C07252=1043.907,204.076,-99.284,170.932,38.862,157.345
C07253=1043.914,204.324,-99.309,170.935,38.863,157.345
C07254=1043.920,204.573,-99.334,170.938,38.865,157.345
C07255=1043.927,204.821,-99.359,170.940,38.867,157.346
C07256=1043.933,205.071,-99.384,170.943,38.868,157.346
C07257=1043.959,206.122,-99.491,171.208,38.971,157.375
C07258=1043.966,206.407,-99.521,171.211,38.973,157.375
C07259=1043.974,206.692,-99.551,171.213,38.976,157.376
C07260=1043.982,206.977,-99.581,171.216,38.979,157.376
C07261=1043.989,207.263,-99.612,171.219,38.982,157.377
C07262=1043.995,207.512,-99.637,171.220,38.984,157.378
C07263=1044.003,207.760,-99.664,171.223,38.987,157.378
C07264=1044.008,208.009,-99.690,171.224,38.989,157.379
C07265=1044.015,208.257,-99.717,171.227,38.992,157.379
C07266=1044.022,208.505,-99.743,171.229,38.994,157.380
C07267=1044.028,208.755,-99.770,171.231,38.997,157.381
C07268=1044.035,209.003,-99.796,171.234,38.999,157.381
C07269=1044.042,209.251,-99.822,171.235,39.002,157.382
C07270=1044.048,209.500,-99.849,171.238,39.004,157.382
C07271=1044.055,209.748,-99.875,171.239,39.007,157.383
C07272=1044.061,209.996,-99.901,171.242,39.009,157.384
C07273=1044.068,210.245,-99.929,171.244,39.012,157.384
C07274=1044.075,210.493,-99.955,171.246,39.014,157.385
C07275=1044.082,210.742,-99.982,171.248,39.017,157.385
C07276=1044.087,210.990,-100.008,171.250,39.019,157.386
C07277=1044.095,211.239,-100.035,171.252,39.022,157.386
C07278=1044.101,211.488,-100.062,171.255,39.024,157.387
C07279=1044.107,211.736,-100.088,171.256,39.027,157.388
C07280=1044.115,211.985,-100.114,171.259,39.029,157.388
C07281=1044.120,212.233,-100.141,171.262,39.032,157.389
C07282=1044.127,212.481,-100.169,171.263,39.035,157.389
C07283=1044.133,212.730,-100.195,171.266,39.037,157.390
C07284=1044.140,212.979,-100.222,171.267,39.039,157.390
C07285=1044.147,213.227,-100.248,171.270,39.042,157.391
C07286=1044.153,213.476,-100.275,171.272,39.044,157.392
C07287=1044.160,213.724,-100.302,171.274,39.047,157.392
C07288=1044.166,213.972,-100.329,171.276,39.049,157.393
C07289=1044.173,214.221,-100.355,171.279,39.052,157.393
C07290=1044.179,214.469,-100.382,171.280,39.054,157.394
C07291=1044.186,214.718,-100.409,171.283,39.057,157.395
C07292=1044.193,214.967,-100.436,171.286,39.059,157.395
C07293=1044.198,215.215,-100.462,171.287,39.062,157.396
C07294=1044.206,215.464,-100.489,171.290,39.064,157.396
C07295=1044.212,215.712,-100.517,171.291,39.067,157.397
C07296=1044.219,215.960,-100.543,171.294,39.069,157.397
C07297=1044.225,216.209,-100.570,171.296,39.072,157.398
C07298=1044.232,216.458,-100.597,171.298,39.074,157.399
C07299=1044.238,216.706,-100.623,171.300,39.077,157.399
C07300=1044.245,216.955,-100.650,171.303,39.079,157.400
C07301=1044.251,217.202,-100.677,171.306,39.082,157.400
C07302=1044.258,217.451,-100.704,171.307,39.084,157.401
C07303=1044.265,217.700,-100.732,171.310,39.087,157.402
C07304=1044.272,217.948,-100.758,171.312,39.089,157.402
C07305=1044.277,218.197,-100.785,171.314,39.091,157.403
C07306=1044.285,218.445,-100.812,171.316,39.094,157.403
C07307=1044.291,218.694,-100.839,171.319,39.096,157.404
C07308=1044.298,218.941,-100.866,171.320,39.099,157.404
C07309=1044.304,219.190,-100.893,171.323,39.101,157.405
C07310=1044.311,219.439,-100.921,171.325,39.103,157.406
C07311=1044.318,219.688,-100.947,171.328,39.106,157.406
C07312=1044.324,219.936,-100.974,171.329,39.109,157.407
C07313=1044.331,220.184,-101.001,171.332,39.111,157.407
C07314=1044.338,220.475,-101.033,171.335,39.114,157.408
C07315=1044.346,220.766,-101.065,171.337,39.117,157.409
C07316=1044.353,221.056,-101.097,171.340,39.120,157.409
C07317=1044.362,221.347,-101.129,171.343,39.123,157.410
C07318=1044.367,221.596,-101.155,171.345,39.125,157.411
C07319=1044.374,221.844,-101.183,171.347,39.128,157.411
C07320=1044.381,222.093,-101.210,171.349,39.130,157.412
C07321=1044.387,222.341,-101.237,171.352,39.133,157.412
C07322=1044.394,222.589,-101.265,171.354,39.135,157.413
C07323=1044.400,222.838,-101.292,171.356,39.138,157.414
C07324=1044.407,223.087,-101.319,171.358,39.140,157.414
C07325=1044.413,223.334,-101.347,171.361,39.142,157.415
C07326=1044.420,223.583,-101.374,171.364,39.145,157.415
C07327=1044.427,223.831,-101.401,171.365,39.148,157.416
C07328=1044.434,224.080,-101.429,171.368,39.150,157.417
C07329=1044.439,224.328,-101.455,171.370,39.152,157.417
C07330=1044.446,224.577,-101.483,171.373,39.155,157.418
C07331=1044.453,224.825,-101.511,171.374,39.158,157.418
C07332=1044.459,225.074,-101.539,171.377,39.160,157.419
C07333=1044.466,225.323,-101.566,171.379,39.162,157.420
C07334=1044.472,225.570,-101.593,171.382,39.164,157.420
C07335=1044.479,225.819,-101.620,171.385,39.167,157.421
C07336=1044.486,226.067,-101.648,171.386,39.170,157.421
C07337=1044.492,226.316,-101.675,171.389,39.172,157.422
C07338=1044.499,226.564,-101.703,171.391,39.174,157.422
C07339=1044.506,226.813,-101.730,171.394,39.177,157.423
C07340=1044.512,227.061,-101.758,171.396,39.179,157.424
C07341=1044.519,227.309,-101.785,171.398,39.182,157.424
C07342=1044.525,227.558,-101.812,171.400,39.184,157.425
C07343=1044.532,227.807,-101.840,171.403,39.186,157.425
C07344=1044.539,228.055,-101.867,171.405,39.189,157.426
C07345=1044.546,228.303,-101.895,171.408,39.192,157.427
C07346=1044.552,228.552,-101.923,171.410,39.194,157.427
C07347=1044.559,228.800,-101.950,171.412,39.196,157.428
C07348=1044.565,229.048,-101.978,171.415,39.199,157.428
C07349=1044.572,229.296,-102.006,171.417,39.201,157.429
C07350=1044.578,229.545,-102.034,171.420,39.204,157.429
C07351=1044.584,229.793,-102.062,171.421,39.206,157.430
C07352=1044.591,230.042,-102.089,171.424,39.208,157.431
C07353=1044.598,230.290,-102.117,171.427,39.211,157.431
C07354=1044.604,230.539,-102.145,171.429,39.214,157.432
C07355=1044.611,230.786,-102.172,171.432,39.216,157.432
C07356=1044.617,231.035,-102.200,171.434,39.218,157.433
C07357=1044.624,231.283,-102.228,171.436,39.221,157.434
C07358=1044.631,231.532,-102.255,171.438,39.223,157.434
C07359=1044.637,231.781,-102.284,171.441,39.226,157.435
C07360=1044.643,232.029,-102.311,171.443,39.228,157.435
C07361=1044.650,232.277,-102.339,171.446,39.231,157.436
C07362=1044.657,232.526,-102.367,171.449,39.233,157.437
C07363=1044.663,232.774,-102.395,171.451,39.236,157.437
C07364=1044.669,233.023,-102.423,171.453,39.238,157.438
C07365=1044.675,233.271,-102.450,171.455,39.241,157.438
C07366=1044.682,233.519,-102.479,171.458,39.243,157.439
C07367=1044.689,233.767,-102.506,171.461,39.246,157.440
C07368=1044.695,234.016,-102.535,171.463,39.248,157.440
C07369=1044.702,234.264,-102.562,171.466,39.251,157.441
C07370=1044.709,234.547,-102.595,171.468,39.253,157.441
C07371=1044.717,234.831,-102.627,171.471,39.256,157.442
C07372=1044.724,235.114,-102.658,171.474,39.259,157.443
C07373=1044.731,235.397,-102.691,171.476,39.262,157.444
C07374=1044.738,235.646,-102.718,171.479,39.264,157.444
C07375=1044.745,235.894,-102.746,171.481,39.267,157.445
C07376=1044.751,236.142,-102.775,171.484,39.269,157.445
C07377=1044.758,236.391,-102.803,171.487,39.272,157.446
C07378=1044.764,236.639,-102.831,171.489,39.274,157.447
C07379=1044.771,236.887,-102.858,171.492,39.276,157.447
C07380=1044.777,237.136,-102.887,171.494,39.279,157.448
C07381=1044.784,237.384,-102.915,171.497,39.282,157.448
C07382=1044.790,237.632,-102.943,171.498,39.284,157.449
C07383=1044.797,237.881,-102.972,171.501,39.286,157.449
C07384=1044.803,238.129,-103.000,171.504,39.289,157.450
C07385=1044.810,238.377,-103.028,171.506,39.291,157.451
C07386=1044.816,238.626,-103.056,171.509,39.294,157.451
C07387=1044.823,238.874,-103.084,171.511,39.296,157.452
C07388=1044.830,239.122,-103.113,171.514,39.299,157.453
C07389=1044.837,239.371,-103.141,171.516,39.301,157.453
C07390=1044.844,239.619,-103.170,171.519,39.303,157.454
C07391=1044.850,239.868,-103.197,171.521,39.306,157.454
C07392=1044.856,240.116,-103.226,171.524,39.309,157.455
C07393=1044.863,240.364,-103.254,171.527,39.311,157.455
C07394=1044.870,240.613,-103.282,171.529,39.313,157.456
C07395=1044.876,240.861,-103.311,171.532,39.315,157.457
C07396=1044.883,241.109,-103.339,171.534,39.318,157.457
C07397=1044.889,241.357,-103.368,171.537,39.321,157.458
C07398=1044.896,241.606,-103.395,171.540,39.323,157.458
C07399=1044.902,241.854,-103.425,171.542,39.326,157.459
C07400=1044.909,242.102,-103.453,171.545,39.328,157.460
C07401=1044.915,242.350,-103.481,171.547,39.330,157.460
C07402=1044.922,242.599,-103.511,171.550,39.333,157.461
C07403=1044.929,242.847,-103.539,171.553,39.335,157.462
C07404=1044.935,243.096,-103.567,171.554,39.338,157.462
C07405=1044.942,243.344,-103.596,171.557,39.341,157.463
C07406=1044.948,243.592,-103.624,171.559,39.343,157.463
C07407=1044.954,243.841,-103.653,171.562,39.345,157.464
C07408=1044.961,244.088,-103.682,171.564,39.348,157.465
C07409=1044.967,244.336,-103.711,171.567,39.350,157.465
C07410=1044.974,244.585,-103.738,171.570,39.353,157.466
C07411=1044.981,244.834,-103.768,171.572,39.355,157.466
C07412=1044.987,245.082,-103.797,171.575,39.358,157.467
C07413=1044.994,245.330,-103.825,171.577,39.360,157.468
C07414=1045.000,245.578,-103.854,171.580,39.363,157.468
C07415=1045.006,245.827,-103.883,171.583,39.365,157.469
C07416=1045.012,246.075,-103.912,171.585,39.368,157.470
C07417=1045.019,246.323,-103.940,171.588,39.370,157.470
C07418=1045.026,246.571,-103.969,171.590,39.373,157.471
C07419=1045.032,246.820,-103.998,171.593,39.375,157.471
C07420=1045.038,247.068,-104.027,171.596,39.378,157.472
C07421=1045.045,247.316,-104.056,171.598,39.381,157.473
C07422=1045.051,247.565,-104.085,171.601,39.383,157.473
C07423=1045.057,247.813,-104.114,171.603,39.386,157.474
C07424=1045.064,248.060,-104.143,171.606,39.388,157.474
C07425=1045.070,248.309,-104.172,171.610,39.390,157.475
C07426=1045.077,248.587,-104.204,171.612,39.393,157.476
C07427=1045.085,248.864,-104.236,171.615,39.396,157.476
C07428=1045.092,249.141,-104.269,171.618,39.399,157.477
C07429=1045.099,249.419,-104.302,171.621,39.402,157.478
C07430=1045.106,249.667,-104.330,171.624,39.405,157.479
C07431=1045.112,249.915,-104.359,171.627,39.407,157.479
C07432=1045.119,250.164,-104.389,171.629,39.409,157.480
C07433=1045.125,250.412,-104.418,171.632,39.412,157.480
C07434=1045.131,250.660,-104.447,171.634,39.414,157.481
C07435=1045.137,250.908,-104.476,171.637,39.417,157.482
C07436=1045.144,251.157,-104.505,171.640,39.419,157.482
C07437=1045.151,251.405,-104.534,171.642,39.422,157.483
C07438=1045.157,251.653,-104.563,171.645,39.424,157.484
C07439=1045.164,251.900,-104.592,171.647,39.427,157.484
C07440=1045.171,252.149,-104.622,171.650,39.430,157.485
C07441=1045.177,252.397,-104.651,171.654,39.432,157.485
C07442=1045.183,252.646,-104.680,171.656,39.434,157.486
C07443=1045.190,252.894,-104.709,171.659,39.437,157.487
C07444=1045.197,253.143,-104.738,171.661,39.439,157.487
C07445=1045.203,253.391,-104.767,171.664,39.442,157.488
C07446=1045.209,253.639,-104.796,171.667,39.444,157.488
C07447=1045.216,253.887,-104.826,171.669,39.447,157.489
C07448=1045.222,254.135,-104.855,171.672,39.449,157.490
C07449=1045.229,254.383,-104.885,171.674,39.452,157.490
C07450=1045.236,254.632,-104.913,171.678,39.454,157.491
C07451=1045.243,254.879,-104.943,171.681,39.457,157.492
C07452=1045.249,255.127,-104.972,171.683,39.459,157.492
C07453=1045.256,255.376,-105.002,171.686,39.462,157.493
C07454=1045.262,255.624,-105.031,171.688,39.464,157.493
C07455=1045.269,255.872,-105.060,171.691,39.466,157.494
C07456=1045.276,256.121,-105.090,171.694,39.469,157.495
C07457=1045.282,256.369,-105.119,171.697,39.471,157.495
C07458=1045.289,256.618,-105.148,171.700,39.474,157.496
C07459=1045.295,256.865,-105.178,171.702,39.477,157.497
C07460=1045.302,257.113,-105.207,171.705,39.479,157.497
C07461=1045.308,257.362,-105.236,171.708,39.482,157.498
C07462=1045.315,257.610,-105.266,171.710,39.484,157.498
C07463=1045.322,257.859,-105.296,171.714,39.486,157.499
C07464=1045.329,258.106,-105.325,171.717,39.489,157.500
C07465=1045.335,258.354,-105.354,171.719,39.491,157.500
C07466=1045.342,258.603,-105.383,171.722,39.494,157.501
C07467=1045.349,258.850,-105.413,171.724,39.496,157.502
C07468=1045.356,259.099,-105.442,171.728,39.498,157.502
C07469=1045.362,259.347,-105.472,171.731,39.501,157.503
C07470=1045.369,259.595,-105.501,171.733,39.504,157.503
C07471=1045.376,259.843,-105.531,171.736,39.506,157.504
C07472=1045.382,260.092,-105.561,171.738,39.509,157.505
C07473=1045.389,260.339,-105.590,171.742,39.511,157.505
C07474=1045.396,260.588,-105.620,171.745,39.513,157.506
C07475=1045.402,260.836,-105.650,171.747,39.516,157.507
C07476=1045.409,261.084,-105.679,171.750,39.518,157.507
C07477=1045.416,261.332,-105.709,171.754,39.521,157.508
C07478=1045.423,261.581,-105.738,171.756,39.523,157.508
C07479=1045.429,261.828,-105.768,171.759,39.525,157.509
C07480=1045.436,262.077,-105.797,171.761,39.528,157.510
C07481=1045.443,262.325,-105.827,171.765,39.530,157.510
C07482=1045.450,262.600,-105.860,171.768,39.533,157.511
C07483=1045.457,262.876,-105.894,171.771,39.536,157.512
C07484=1045.465,263.153,-105.926,171.774,39.539,157.513
C07485=1045.472,263.429,-105.960,171.778,39.542,157.513
C07486=1045.479,263.677,-105.990,171.780,39.545,157.514
C07487=1045.485,263.925,-106.020,171.783,39.547,157.515
C07488=1045.492,264.173,-106.050,171.786,39.550,157.515
C07489=1045.498,264.421,-106.079,171.788,39.552,157.516
C07490=1045.505,264.670,-106.110,171.792,39.555,157.517
C07491=1045.511,264.917,-106.140,171.794,39.557,157.517
C07492=1045.518,265.165,-106.170,171.797,39.560,157.518
C07493=1045.524,265.413,-106.200,171.801,39.563,157.519
C07494=1045.531,265.662,-106.230,171.803,39.565,157.519
C07495=1045.537,265.910,-106.259,171.806,39.568,157.520
C07496=1045.544,266.158,-106.290,171.809,39.570,157.520
C07497=1045.551,266.406,-106.320,171.812,39.573,157.521
C07498=1045.558,266.654,-106.350,171.815,39.575,157.522
C07499=1045.564,266.902,-106.381,171.818,39.578,157.522
C07500=1045.571,267.150,-106.411,171.820,39.580,157.523
C07501=1045.578,267.398,-106.441,171.824,39.583,157.524
C07502=1045.584,267.647,-106.471,171.827,39.585,157.524
C07503=1045.591,267.894,-106.501,171.829,39.588,157.525
C07504=1045.597,268.143,-106.532,171.833,39.591,157.526
C07505=1045.604,268.390,-106.562,171.836,39.593,157.526
C07506=1045.610,268.639,-106.592,171.838,39.596,157.527
C07507=1045.617,268.886,-106.622,171.842,39.598,157.528
C07508=1045.623,269.135,-106.653,171.845,39.601,157.528
C07509=1045.630,269.383,-106.683,171.847,39.603,157.529
C07510=1045.636,269.631,-106.713,171.851,39.606,157.530
C07511=1045.643,269.879,-106.743,171.854,39.609,157.530
C07512=1045.650,270.127,-106.774,171.856,39.611,157.531
C07513=1045.656,270.375,-106.804,171.859,39.614,157.532
C07514=1045.663,270.624,-106.835,171.863,39.616,157.532
C07515=1045.670,270.872,-106.865,171.865,39.619,157.533
C07516=1045.676,271.119,-106.896,171.869,39.621,157.534
C07517=1045.683,271.367,-106.926,171.871,39.624,157.534
C07518=1045.689,271.616,-106.957,171.874,39.626,157.535
C07519=1045.696,271.863,-106.986,171.878,39.629,157.536
C07520=1045.702,272.112,-107.017,171.880,39.631,157.536
C07521=1045.709,272.360,-107.048,171.883,39.634,157.537
C07522=1045.716,272.607,-107.078,171.887,39.637,157.538
C07523=1045.722,272.856,-107.109,171.889,39.639,157.538
C07524=1045.729,273.104,-107.140,171.892,39.642,157.539
C07525=1045.735,273.351,-107.170,171.896,39.645,157.540
C07526=1045.742,273.600,-107.201,171.898,39.647,157.540
C07527=1045.748,273.848,-107.232,171.901,39.650,157.541
C07528=1045.755,274.095,-107.262,171.905,39.653,157.542
C07529=1045.762,274.344,-107.293,171.907,39.655,157.542
C07530=1045.768,274.592,-107.323,171.911,39.658,157.543
C07531=1045.775,274.840,-107.354,171.914,39.660,157.544
C07532=1045.781,275.087,-107.385,171.916,39.663,157.544
C07533=1045.788,275.336,-107.415,171.920,39.665,157.545
C07534=1045.794,275.584,-107.447,171.923,39.668,157.546
C07535=1045.802,275.832,-107.477,171.927,39.671,157.547
C07536=1045.808,276.079,-107.508,171.929,39.673,157.547
C07537=1045.814,276.328,-107.539,171.932,39.676,157.548
C07538=1045.825,276.739,-107.590,171.937,39.681,157.549
C07539=1045.832,276.982,-107.620,171.941,39.683,157.550
C07540=1045.838,277.225,-107.650,171.943,39.686,157.550
C07541=1045.845,277.468,-107.681,171.946,39.688,157.551
C07542=1045.851,277.711,-107.711,171.950,39.691,157.552
C07543=1045.858,277.954,-107.742,171.952,39.693,157.552
C07544=1045.865,278.198,-107.772,171.956,39.696,157.553
C07545=1045.871,278.441,-107.802,171.959,39.698,157.554
C07546=1045.877,278.690,-107.833,171.961,39.701,157.554
C07547=1045.884,278.937,-107.864,171.965,39.704,157.555
C07548=1045.891,279.185,-107.895,171.968,39.707,157.556
C07549=1045.897,279.433,-107.926,171.971,39.709,157.557
C07550=1045.904,279.681,-107.957,171.974,39.712,157.557
C07551=1045.911,279.929,-107.989,171.978,39.714,157.558
C07552=1045.917,280.177,-108.019,171.980,39.717,157.559
C07553=1045.923,280.425,-108.050,171.984,39.720,157.559
C07554=1045.930,280.672,-108.082,171.987,39.723,157.560
C07555=1045.937,280.920,-108.113,171.990,39.726,157.561
C07556=1045.943,281.169,-108.144,171.993,39.728,157.561
C07557=1045.950,281.417,-108.175,171.996,39.731,157.562
C07558=1045.957,281.665,-108.207,172.000,39.733,157.563
C07559=1045.963,281.912,-108.238,172.002,39.736,157.564
C07560=1045.969,282.160,-108.270,172.006,39.739,157.564
C07561=1045.976,282.408,-108.301,172.009,39.742,157.565
C07562=1045.982,282.657,-108.332,172.013,39.744,157.566
C07563=1045.989,282.904,-108.363,172.015,39.747,157.566
C07564=1045.995,283.152,-108.395,172.019,39.749,157.567
C07565=1046.002,283.400,-108.426,172.022,39.752,157.568
C07566=1046.009,283.648,-108.458,172.025,39.755,157.568
C07567=1046.016,283.896,-108.489,172.028,39.758,157.569
C07568=1046.022,284.144,-108.521,172.032,39.760,157.570
C07569=1046.029,284.392,-108.552,172.035,39.763,157.571
C07570=1046.036,284.640,-108.584,172.038,39.766,157.571
C07571=1046.043,284.888,-108.615,172.041,39.769,157.572
C07572=1046.049,285.136,-108.646,172.045,39.772,157.573
C07573=1046.056,285.383,-108.678,172.047,39.774,157.573
C07574=1046.063,285.631,-108.709,172.051,39.776,157.574
C07575=1046.069,285.879,-108.741,172.055,39.779,157.575
C07576=1046.076,286.127,-108.772,172.058,39.782,157.576
C07577=1046.083,286.375,-108.804,172.061,39.785,157.576
C07578=1046.090,286.623,-108.835,172.064,39.788,157.577
C07579=1046.096,286.871,-108.866,172.068,39.790,157.578
C07580=1046.103,287.119,-108.898,172.070,39.793,157.579
C07581=1046.110,287.367,-108.929,172.074,39.796,157.579
C07582=1046.116,287.615,-108.961,172.078,39.799,157.580
C07583=1046.123,287.862,-108.993,172.081,39.801,157.581
C07584=1046.130,288.110,-109.025,172.084,39.804,157.581
C07585=1046.136,288.358,-109.056,172.087,39.807,157.582
C07586=1046.142,288.606,-109.088,172.091,39.810,157.583
C07587=1046.149,288.853,-109.120,172.094,39.812,157.584
C07588=1046.156,289.101,-109.152,172.097,39.815,157.584
C07589=1046.163,289.349,-109.183,172.101,39.818,157.585
C07590=1046.169,289.598,-109.215,172.104,39.821,157.586
C07591=1046.176,289.845,-109.248,172.108,39.823,157.587
C07592=1046.182,290.093,-109.279,172.110,39.826,157.587
C07593=1046.189,290.341,-109.310,172.114,39.829,157.588
C07594=1046.197,290.633,-109.348,172.118,39.832,157.589
C07595=1046.205,290.924,-109.387,172.122,39.835,157.590
C07596=1046.212,291.216,-109.424,172.126,39.839,157.591
C07597=1046.220,291.509,-109.462,172.130,39.842,157.592
C07598=1046.227,291.757,-109.494,172.133,39.845,157.592
C07599=1046.234,292.004,-109.526,172.136,39.848,157.593
C07600=1046.240,292.252,-109.558,172.140,39.850,157.594
C07601=1046.247,292.500,-109.590,172.144,39.853,157.595
C07602=1046.254,292.748,-109.621,172.146,39.856,157.595
C07603=1046.260,292.995,-109.654,172.150,39.859,157.596
C07604=1046.268,293.244,-109.686,172.154,39.862,157.597
C07605=1046.275,293.491,-109.718,172.157,39.865,157.598
C07606=1046.281,293.739,-109.750,172.160,39.867,157.598
C07607=1046.288,293.987,-109.782,172.164,39.870,157.599
C07608=1046.294,294.235,-109.814,172.167,39.873,157.600
C07609=1046.301,294.482,-109.846,172.171,39.876,157.601
C07610=1046.308,294.730,-109.879,172.174,39.878,157.601
C07611=1046.314,294.978,-109.911,172.177,39.882,157.602
C07612=1046.321,295.226,-109.944,172.181,39.884,157.603
C07613=1046.328,295.473,-109.976,172.185,39.887,157.604
C07614=1046.334,295.721,-110.007,172.187,39.890,157.604
C07615=1046.341,295.969,-110.040,172.191,39.893,157.605
C07616=1046.348,296.217,-110.073,172.195,39.896,157.606
C07617=1046.354,296.465,-110.106,172.198,39.899,157.607
C07618=1046.361,296.712,-110.137,172.202,39.901,157.607
C07619=1046.367,296.960,-110.170,172.206,39.905,157.608
C07620=1046.373,297.208,-110.203,172.208,39.908,157.609
C07621=1046.380,297.456,-110.236,172.212,39.910,157.610
C07622=1046.386,297.703,-110.269,172.216,39.914,157.611
C07623=1046.393,297.951,-110.301,172.219,39.916,157.611
C07624=1046.400,298.198,-110.333,172.223,39.920,157.612
C07625=1046.407,298.447,-110.367,172.226,39.922,157.613
C07626=1046.413,298.695,-110.399,172.229,39.925,157.614
C07627=1046.420,298.942,-110.431,172.233,39.928,157.615
C07628=1046.426,299.190,-110.463,172.237,39.931,157.615
C07629=1046.433,299.438,-110.497,172.241,39.934,157.616
C07630=1046.439,299.686,-110.529,172.243,39.937,157.617
C07631=1046.445,299.933,-110.562,172.247,39.940,157.618
C07632=1046.452,300.180,-110.594,172.251,39.943,157.619
C07633=1046.459,300.429,-110.627,172.254,39.946,157.619
C07634=1046.466,300.676,-110.661,172.258,39.949,157.620
C07635=1046.472,300.923,-110.694,172.261,39.952,157.621
C07636=1046.479,301.172,-110.727,172.265,39.955,157.622
C07637=1046.485,301.419,-110.759,172.268,39.958,157.623
C07638=1046.492,301.667,-110.792,172.272,39.961,157.623
C07639=1046.499,301.915,-110.825,172.276,39.964,157.624
C07640=1046.506,302.162,-110.857,172.279,39.967,157.625
C07641=1046.512,302.410,-110.890,172.282,39.970,157.626
C07642=1046.519,302.658,-110.923,172.286,39.973,157.627
C07643=1046.525,302.905,-110.957,172.290,39.975,157.627
C07644=1046.532,303.153,-110.989,172.294,39.979,157.628
C07645=1046.539,303.401,-111.022,172.298,39.981,157.629
C07646=1046.546,303.648,-111.055,172.300,39.985,157.630
C07647=1046.553,303.896,-111.088,172.304,39.987,157.631
C07648=1046.559,304.144,-111.121,172.308,39.991,157.632
C07649=1046.565,304.391,-111.154,172.312,39.993,157.632
C07650=1046.575,304.699,-111.195,172.316,39.997,157.633
C07651=1046.582,305.008,-111.236,172.321,40.001,157.634
C07652=1046.591,305.316,-111.277,172.325,40.005,157.635
C07653=1046.600,305.624,-111.319,172.330,40.009,157.636
C07654=1046.606,305.872,-111.352,172.334,40.011,157.637
C07655=1046.613,306.120,-111.385,172.338,40.015,157.638
C07656=1046.620,306.367,-111.418,172.341,40.017,157.639
C07657=1046.627,306.615,-111.451,172.344,40.021,157.640
C07658=1046.634,306.862,-111.484,172.348,40.023,157.640
C07659=1046.641,307.111,-111.518,172.352,40.027,157.641
C07660=1046.647,307.358,-111.550,172.356,40.029,157.642
C07661=1046.654,307.606,-111.584,172.360,40.033,157.643
C07662=1046.661,307.853,-111.617,172.364,40.035,157.644
C07663=1046.668,308.101,-111.651,172.368,40.039,157.645
C07664=1046.675,308.348,-111.683,172.370,40.042,157.646
C07665=1046.682,308.596,-111.717,172.374,40.045,157.646
C07666=1046.689,308.844,-111.750,172.378,40.048,157.647
C07667=1046.696,309.091,-111.783,172.382,40.051,157.648
C07668=1046.703,309.339,-111.817,172.386,40.054,157.649
C07669=1046.709,309.587,-111.850,172.390,40.057,157.650
C07670=1046.716,309.834,-111.884,172.393,40.060,157.650
C07671=1046.723,310.082,-111.917,172.397,40.063,157.651
C07672=1046.730,310.330,-111.950,172.401,40.066,157.652
C07673=1046.737,310.577,-111.984,172.405,40.069,157.653
C07674=1046.744,310.826,-112.017,172.409,40.072,157.654
C07675=1046.751,311.072,-112.050,172.412,40.075,157.655
C07676=1046.758,311.320,-112.084,172.416,40.078,157.656
C07677=1046.766,311.568,-112.118,172.420,40.082,157.656
C07678=1046.772,311.815,-112.150,172.423,40.084,157.657
C07679=1046.779,312.063,-112.184,172.427,40.087,157.658
C07680=1046.786,312.310,-112.218,172.431,40.091,157.659
C07681=1046.794,312.558,-112.252,172.435,40.093,157.660
C07682=1046.800,312.806,-112.285,172.439,40.097,157.661
C07683=1046.806,313.054,-112.319,172.443,40.100,157.662
C07684=1046.813,313.301,-112.353,172.447,40.103,157.662
C07685=1046.819,313.549,-112.387,172.451,40.106,157.663
C07686=1046.827,313.796,-112.421,172.455,40.110,157.664
C07687=1046.834,314.044,-112.454,172.459,40.113,157.665
C07688=1046.840,314.291,-112.489,172.462,40.116,157.666
C07689=1046.847,314.539,-112.522,172.466,40.119,157.667
C07690=1046.854,314.786,-112.558,172.470,40.123,157.668
C07691=1046.860,315.033,-112.591,172.474,40.126,157.669
C07692=1046.867,315.281,-112.625,172.477,40.129,157.670
C07693=1046.874,315.529,-112.659,172.481,40.133,157.670
C07694=1046.880,315.776,-112.693,172.485,40.136,157.671
C07695=1046.887,316.024,-112.727,172.489,40.139,157.672
C07696=1046.893,316.272,-112.762,172.493,40.142,157.673
C07697=1046.901,316.520,-112.795,172.497,40.146,157.674
C07698=1046.907,316.766,-112.830,172.501,40.149,157.675
C07699=1046.914,317.014,-112.864,172.505,40.152,157.676
C07700=1046.920,317.262,-112.898,172.509,40.155,157.677
C07701=1046.928,317.510,-112.932,172.513,40.159,157.678
C07702=1046.934,317.758,-112.967,172.516,40.162,157.679
C07703=1046.941,318.004,-113.001,172.520,40.165,157.679
C07704=1046.947,318.252,-113.035,172.524,40.168,157.680
C07705=1046.955,318.500,-113.069,172.528,40.172,157.681
C07706=1046.963,318.812,-113.113,172.534,40.176,157.682
C07707=1046.971,319.125,-113.156,172.539,40.180,157.684
C07708=1046.980,319.438,-113.200,172.544,40.184,157.685
C07709=1046.989,319.751,-113.243,172.549,40.188,157.686
C07710=1046.996,319.999,-113.277,172.553,40.191,157.687
C07711=1047.003,320.246,-113.312,172.557,40.195,157.688
C07712=1047.010,320.494,-113.346,172.561,40.198,157.689
C07713=1047.016,320.740,-113.381,172.565,40.202,157.690
C07714=1047.023,320.988,-113.415,172.569,40.205,157.691
C07715=1047.030,321.235,-113.449,172.573,40.208,157.691
C07716=1047.037,321.483,-113.484,172.577,40.212,157.692
C07717=1047.044,321.730,-113.519,172.581,40.215,157.693
C07718=1047.051,321.978,-113.553,172.585,40.218,157.694
C07719=1047.058,322.226,-113.588,172.589,40.222,157.695
C07720=1047.065,322.473,-113.622,172.593,40.225,157.696
C07721=1047.072,322.721,-113.657,172.598,40.228,157.697
C07722=1047.079,322.968,-113.691,172.602,40.231,157.698
C07723=1047.086,323.216,-113.726,172.606,40.235,157.699
C07724=1047.092,323.463,-113.761,172.610,40.238,157.700
C07725=1047.100,323.711,-113.795,172.614,40.242,157.701
C07726=1047.106,323.958,-113.830,172.618,40.245,157.702
C07727=1047.114,324.206,-113.865,172.622,40.248,157.703
C07728=1047.121,324.454,-113.899,172.626,40.252,157.704
C07729=1047.128,324.701,-113.934,172.631,40.255,157.705
C07730=1047.135,324.948,-113.969,172.635,40.258,157.705
C07731=1047.142,325.196,-114.003,172.639,40.262,157.707
C07732=1047.149,325.443,-114.038,172.643,40.265,157.707
C07733=1047.156,325.691,-114.073,172.647,40.269,157.708
C07734=1047.163,325.938,-114.108,172.651,40.272,157.709
C07735=1047.170,326.185,-114.143,172.656,40.275,157.710
C07736=1047.177,326.434,-114.178,172.660,40.279,157.711
C07737=1047.185,326.681,-114.212,172.664,40.283,157.712
C07738=1047.192,326.928,-114.247,172.668,40.286,157.713
C07739=1047.198,327.175,-114.282,172.672,40.289,157.714
C07740=1047.206,327.422,-114.317,172.677,40.293,157.715
C07741=1047.213,327.671,-114.352,172.681,40.296,157.716
C07742=1047.220,327.918,-114.388,172.685,40.300,157.717
C07743=1047.227,328.165,-114.422,172.689,40.303,157.718
C07744=1047.234,328.412,-114.457,172.693,40.306,157.719
C07745=1047.242,328.660,-114.492,172.698,40.310,157.720
C07746=1047.249,328.907,-114.527,172.702,40.313,157.721
C07747=1047.256,329.155,-114.562,172.706,40.317,157.722
C07748=1047.263,329.402,-114.597,172.710,40.320,157.723
C07749=1047.271,329.650,-114.632,172.715,40.324,157.724
C07750=1047.277,329.897,-114.668,172.719,40.327,157.725
C07751=1047.284,330.145,-114.703,172.723,40.331,157.726
C07752=1047.291,330.392,-114.738,172.727,40.335,157.727
C07753=1047.299,330.639,-114.774,172.732,40.338,157.728
C07754=1047.305,330.887,-114.809,172.736,40.341,157.729
C07755=1047.312,331.134,-114.844,172.740,40.345,157.730
C07756=1047.319,331.382,-114.879,172.744,40.349,157.731
C07757=1047.327,331.629,-114.916,172.748,40.352,157.732
C07758=1047.333,331.876,-114.951,172.753,40.356,157.733
C07759=1047.339,332.124,-114.987,172.758,40.360,157.734
C07760=1047.347,332.372,-115.023,172.762,40.363,157.735
C07761=1047.354,332.619,-115.058,172.767,40.367,157.736
C07762=1047.362,332.926,-115.102,172.772,40.371,157.737
C07763=1047.371,333.235,-115.146,172.777,40.376,157.739
C07764=1047.381,333.542,-115.191,172.783,40.381,157.740
C07765=1047.389,333.850,-115.235,172.788,40.385,157.741
C07766=1047.396,334.098,-115.270,172.792,40.389,157.742
C07767=1047.403,334.345,-115.306,172.797,40.392,157.743
C07768=1047.410,334.592,-115.341,172.802,40.396,157.744
C07769=1047.418,334.839,-115.378,172.805,40.399,157.745
C07770=1047.425,335.087,-115.413,172.811,40.403,157.746
C07771=1047.432,335.334,-115.449,172.815,40.407,157.747
C07772=1047.439,335.581,-115.485,172.819,40.411,157.748
C07773=1047.447,335.829,-115.520,172.824,40.414,157.750
C07774=1047.454,336.076,-115.556,172.828,40.418,157.751
C07775=1047.460,336.323,-115.593,172.832,40.422,157.752
C07776=1047.468,336.571,-115.628,172.837,40.425,157.753
C07777=1047.475,336.818,-115.664,172.842,40.429,157.754
C07778=1047.482,337.065,-115.701,172.846,40.433,157.755
C07779=1047.488,337.313,-115.736,172.851,40.437,157.756
C07780=1047.496,337.560,-115.772,172.855,40.440,157.757
C07781=1047.502,337.807,-115.809,172.859,40.444,157.758
C07782=1047.510,338.055,-115.845,172.864,40.448,157.759
C07783=1047.517,338.301,-115.881,172.868,40.452,157.760
C07784=1047.524,338.549,-115.917,172.873,40.456,157.761
C07785=1047.531,338.797,-115.953,172.878,40.460,157.763
C07786=1047.538,339.044,-115.989,172.882,40.463,157.764
C07787=1047.546,339.291,-116.025,172.887,40.467,157.765
C07788=1047.552,339.539,-116.061,172.891,40.471,157.766
C07789=1047.560,339.785,-116.097,172.896,40.475,157.767
C07790=1047.567,340.033,-116.133,172.901,40.479,157.768
C07791=1047.574,340.280,-116.170,172.905,40.483,157.769
C07792=1047.581,340.527,-116.206,172.910,40.486,157.770
C07793=1047.589,340.775,-116.242,172.914,40.490,157.771
C07794=1047.596,341.022,-116.279,172.919,40.494,157.772
C07795=1047.603,341.269,-116.315,172.924,40.498,157.773
C07796=1047.610,341.517,-116.352,172.929,40.502,157.775
C07797=1047.617,341.764,-116.388,172.933,40.505,157.776
C07798=1047.625,342.010,-116.425,172.938,40.509,157.777
C07799=1047.632,342.258,-116.461,172.942,40.513,157.778
C07800=1047.640,342.506,-116.498,172.946,40.517,157.779
C07801=1047.646,342.753,-116.534,172.952,40.521,157.780
C07802=1047.654,343.000,-116.570,172.956,40.525,157.781
C07803=1047.661,343.247,-116.608,172.961,40.529,157.782
C07804=1047.668,343.494,-116.644,172.965,40.533,157.784
C07805=1047.675,343.742,-116.681,172.970,40.537,157.785
C07806=1047.683,343.989,-116.717,172.975,40.541,157.786
C07807=1047.689,344.236,-116.754,172.980,40.545,157.787
C07808=1047.696,344.483,-116.791,172.984,40.549,157.788
C07809=1047.704,344.730,-116.828,172.989,40.553,157.789
C07810=1047.711,344.978,-116.864,172.994,40.557,157.790
C07811=1047.718,345.224,-116.901,172.999,40.561,157.792
C07812=1047.725,345.472,-116.938,173.003,40.565,157.793
C07813=1047.733,345.719,-116.975,173.009,40.569,157.794
C07814=1047.740,345.967,-117.012,173.013,40.573,157.795
C07815=1047.747,346.213,-117.049,173.018,40.577,157.796
C07816=1047.754,346.461,-117.086,173.023,40.581,157.797
C07817=1047.762,346.708,-117.122,173.027,40.585,157.799
C07818=1047.770,347.012,-117.168,173.033,40.591,157.800
C07819=1047.780,347.316,-117.214,173.040,40.595,157.802
C07820=1047.788,347.619,-117.260,173.045,40.601,157.803
C07821=1047.797,347.923,-117.304,173.052,40.605,157.804
C07822=1047.804,348.170,-117.342,173.056,40.610,157.806
C07823=1047.812,348.417,-117.379,173.061,40.614,157.807
C07824=1047.819,348.665,-117.415,173.066,40.618,157.808
C07825=1047.826,348.912,-117.453,173.071,40.622,157.809
C07826=1047.834,349.159,-117.491,173.076,40.626,157.810
C07827=1047.842,349.406,-117.527,173.081,40.630,157.812
C07828=1047.848,349.654,-117.564,173.086,40.635,157.813
C07829=1047.856,349.901,-117.602,173.090,40.638,157.814
C07830=1047.864,350.148,-117.639,173.095,40.642,157.815
C07831=1047.871,350.395,-117.676,173.101,40.647,157.816
C07832=1047.878,350.642,-117.714,173.105,40.651,157.818
C07833=1047.885,350.889,-117.751,173.110,40.655,157.819
C07834=1047.893,351.136,-117.789,173.116,40.659,157.820
C07835=1047.900,351.383,-117.826,173.120,40.664,157.821
C07836=1047.907,351.631,-117.864,173.125,40.668,157.823
C07837=1047.914,351.878,-117.901,173.131,40.672,157.824
C07838=1047.922,352.125,-117.939,173.135,40.676,157.825
C07839=1047.929,352.372,-117.976,173.140,40.681,157.826
C07840=1047.936,352.619,-118.014,173.146,40.685,157.828
C07841=1047.944,352.865,-118.052,173.150,40.690,157.829
C07842=1047.952,353.112,-118.089,173.156,40.694,157.830
C07843=1047.959,353.360,-118.127,173.161,40.698,157.831
C07844=1047.966,353.607,-118.164,173.165,40.702,157.833
C07845=1047.973,353.854,-118.202,173.171,40.706,157.834
C07846=1047.981,354.100,-118.240,173.176,40.711,157.835
C07847=1047.988,354.348,-118.278,173.182,40.715,157.837
C07848=1047.995,354.595,-118.315,173.186,40.720,157.838
C07849=1048.003,354.842,-118.353,173.191,40.724,157.839
C07850=1048.010,355.088,-118.391,173.197,40.728,157.840
C07851=1048.018,355.336,-118.429,173.202,40.733,157.842
C07852=1048.026,355.583,-118.467,173.206,40.737,157.843
C07853=1048.033,355.830,-118.505,173.212,40.741,157.844
C07854=1048.040,356.077,-118.542,173.217,40.746,157.846
C07855=1048.048,356.323,-118.580,173.223,40.750,157.847
C07856=1048.056,356.571,-118.618,173.227,40.754,157.848
C07857=1048.063,356.818,-118.656,173.233,40.759,157.849
C07858=1048.070,357.065,-118.694,173.238,40.763,157.851
C07859=1048.078,357.311,-118.732,173.243,40.768,157.852
C07860=1048.084,357.559,-118.770,173.249,40.772,157.853
C07861=1048.093,357.806,-118.809,173.253,40.777,157.855
C07862=1048.100,358.053,-118.847,173.259,40.781,157.856
C07863=1048.107,358.300,-118.885,173.264,40.786,157.857
C07864=1048.115,358.546,-118.923,173.270,40.790,157.859
C07865=1048.123,358.793,-118.962,173.275,40.795,157.860
C07866=1048.130,359.040,-119.000,173.280,40.800,157.861
C07867=1048.137,359.287,-119.038,173.285,40.804,157.863
C07868=1048.145,359.535,-119.077,173.291,40.809,157.864
C07869=1048.153,359.781,-119.115,173.296,40.813,157.865
C07870=1048.160,360.028,-119.153,173.302,40.818,157.867
C07871=1048.168,360.275,-119.192,173.307,40.822,157.868
C07872=1048.175,360.522,-119.230,173.313,40.827,157.869
C07873=1048.183,360.769,-119.268,173.317,40.831,157.871
C07874=1048.193,361.078,-119.317,173.324,40.837,157.872
C07875=1048.201,361.387,-119.365,173.331,40.843,157.874
C07876=1048.211,361.697,-119.413,173.338,40.849,157.876
C07877=1048.221,362.007,-119.462,173.345,40.855,157.878
C07878=1048.228,362.253,-119.500,173.350,40.859,157.879
C07879=1048.236,362.500,-119.539,173.356,40.864,157.880
C07880=1048.243,362.747,-119.578,173.361,40.868,157.882
C07881=1048.251,362.994,-119.616,173.367,40.873,157.883
C07882=1048.259,363.241,-119.655,173.372,40.878,157.885
C07883=1048.266,363.488,-119.693,173.377,40.883,157.886
C07884=1048.274,363.734,-119.733,173.382,40.887,157.887
C07885=1048.281,363.981,-119.772,173.388,40.892,157.889
C07886=1048.288,364.229,-119.811,173.394,40.897,157.890
C07887=1048.296,364.475,-119.849,173.399,40.902,157.892
C07888=1048.304,364.722,-119.889,173.405,40.907,157.893
C07889=1048.311,364.969,-119.927,173.410,40.912,157.895
C07890=1048.319,365.216,-119.966,173.416,40.916,157.896
C07891=1048.327,365.462,-120.005,173.421,40.921,157.897
C07892=1048.334,365.709,-120.045,173.427,40.926,157.899
C07893=1048.342,365.955,-120.084,173.433,40.931,157.900
C07894=1048.349,366.203,-120.123,173.438,40.936,157.902
C07895=1048.358,366.449,-120.162,173.444,40.940,157.903
C07896=1048.365,366.696,-120.201,173.450,40.946,157.905
C07897=1048.373,366.943,-120.240,173.455,40.950,157.906
C07898=1048.380,367.190,-120.279,173.461,40.955,157.907
C07899=1048.388,367.437,-120.319,173.466,40.960,157.909
C07900=1048.396,367.683,-120.358,173.472,40.965,157.910
C07901=1048.403,367.930,-120.397,173.478,40.970,157.912
C07902=1048.411,368.177,-120.436,173.483,40.975,157.913
C07903=1048.419,368.424,-120.476,173.489,40.980,157.915
C07904=1048.427,368.670,-120.515,173.496,40.985,157.916
C07905=1048.434,368.917,-120.555,173.501,40.989,157.918
C07906=1048.442,369.164,-120.594,173.507,40.995,157.919
C07907=1048.450,369.410,-120.634,173.513,41.000,157.921
C07908=1048.457,369.657,-120.673,173.518,41.005,157.922
C07909=1048.466,369.904,-120.712,173.524,41.010,157.924
C07910=1048.473,370.151,-120.752,173.530,41.014,157.925
C07911=1048.481,370.398,-120.792,173.535,41.020,157.927
C07912=1048.489,370.644,-120.831,173.541,41.025,157.929
C07913=1048.497,370.890,-120.871,173.548,41.029,157.930
C07914=1048.505,371.137,-120.910,173.554,41.035,157.932
C07915=1048.513,371.384,-120.950,173.559,41.040,157.933
C07916=1048.521,371.631,-120.990,173.565,41.045,157.935
C07917=1048.528,371.878,-121.030,173.571,41.050,157.936
C07918=1048.535,372.124,-121.069,173.576,41.055,157.938
C07919=1048.543,372.371,-121.109,173.583,41.060,157.939
C07920=1048.551,372.618,-121.149,173.589,41.065,157.941
C07921=1048.560,372.864,-121.189,173.595,41.071,157.942
C07922=1048.567,373.111,-121.229,173.600,41.076,157.944
C07923=1048.575,373.358,-121.269,173.606,41.081,157.946
C07924=1048.582,373.604,-121.309,173.612,41.086,157.947
C07925=1048.590,373.850,-121.349,173.619,41.091,157.949
C07926=1048.598,374.097,-121.389,173.625,41.097,157.950
C07927=1048.606,374.344,-121.429,173.630,41.102,157.952
C07928=1048.614,374.590,-121.470,173.636,41.108,157.954
C07929=1048.621,374.837,-121.510,173.643,41.113,157.955
C07930=1048.632,375.165,-121.564,173.650,41.120,157.957
C07931=1048.643,375.494,-121.617,173.659,41.127,157.959
C07932=1048.654,375.823,-121.670,173.667,41.134,157.962
C07933=1048.664,376.151,-121.724,173.675,41.141,157.964
C07934=1048.671,376.398,-121.764,173.682,41.147,157.965
C07935=1048.680,376.645,-121.805,173.687,41.152,157.967
C07936=1048.688,376.891,-121.845,173.693,41.157,157.969
C07937=1048.696,377.138,-121.885,173.700,41.163,157.970
C07938=1048.704,377.384,-121.926,173.706,41.168,157.972
C07939=1048.712,377.630,-121.967,173.712,41.173,157.973
C07940=1048.720,377.877,-122.007,173.719,41.179,157.975
C07941=1048.728,378.124,-122.047,173.725,41.184,157.977
C07942=1048.736,378.370,-122.088,173.731,41.190,157.979
C07943=1048.744,378.616,-122.129,173.737,41.195,157.980
C07944=1048.752,378.863,-122.170,173.743,41.200,157.982
C07945=1048.760,379.110,-122.209,173.749,41.206,157.984
C07946=1048.768,379.356,-122.250,173.756,41.211,157.985
C07947=1048.776,379.603,-122.291,173.762,41.217,157.987
C07948=1048.785,379.850,-122.332,173.769,41.223,157.989
C07949=1048.793,380.096,-122.372,173.775,41.228,157.990
C07950=1048.800,380.343,-122.414,173.781,41.234,157.992
C07951=1048.808,380.589,-122.454,173.788,41.239,157.994
C07952=1048.816,380.834,-122.496,173.794,41.245,157.996
C07953=1048.825,381.081,-122.537,173.801,41.251,157.997
C07954=1048.832,381.328,-122.578,173.807,41.256,157.999
C07955=1048.840,381.574,-122.618,173.814,41.262,158.001
C07956=1048.848,381.821,-122.659,173.820,41.268,158.003
C07957=1048.857,382.067,-122.701,173.826,41.273,158.004
C07958=1048.865,382.314,-122.742,173.833,41.279,158.006
C07959=1048.873,382.560,-122.783,173.839,41.285,158.008
C07960=1048.881,382.807,-122.825,173.846,41.290,158.010
C07961=1048.889,383.053,-122.866,173.852,41.296,158.011
C07962=1048.897,383.299,-122.906,173.859,41.302,158.013
C07963=1048.906,383.546,-122.948,173.865,41.307,158.015
C07964=1048.913,383.792,-122.989,173.872,41.314,158.017
C07965=1048.921,384.038,-123.030,173.878,41.319,158.018
C07966=1048.930,384.285,-123.071,173.885,41.325,158.020
C07967=1048.938,384.531,-123.113,173.891,41.331,158.022
C07968=1048.946,384.778,-123.154,173.898,41.337,158.024
C07969=1048.954,385.024,-123.196,173.905,41.342,158.026
C07970=1048.963,385.270,-123.238,173.911,41.348,158.027
C07971=1048.971,385.516,-123.279,173.918,41.354,158.029
C07972=1048.979,385.763,-123.321,173.924,41.360,158.031
C07973=1048.987,386.009,-123.362,173.932,41.366,158.033
C07974=1048.996,386.256,-123.403,173.939,41.372,158.035
C07975=1049.004,386.502,-123.445,173.945,41.378,158.037
C07976=1049.012,386.748,-123.487,173.952,41.384,158.038
C07977=1049.021,386.994,-123.528,173.958,41.390,158.040
C07978=1049.029,387.240,-123.571,173.965,41.395,158.042
C07979=1049.038,387.487,-123.612,173.972,41.402,158.044
C07980=1049.046,387.733,-123.653,173.979,41.408,158.046
C07981=1049.054,387.980,-123.695,173.986,41.413,158.048
C07982=1049.063,388.226,-123.737,173.993,41.419,158.050
C07983=1049.071,388.472,-123.779,174.000,41.426,158.052
C07984=1049.080,388.718,-123.821,174.006,41.432,158.054
C07985=1049.089,388.965,-123.862,174.013,41.437,158.055
C07986=1049.100,389.326,-123.924,174.024,41.447,158.058
C07987=1049.113,389.687,-123.987,174.034,41.456,158.061
C07988=1049.125,390.048,-124.048,174.044,41.465,158.064
C07989=1049.137,390.410,-124.110,174.055,41.474,158.067
C07990=1049.146,390.656,-124.152,174.061,41.480,158.069
C07991=1049.154,390.902,-124.195,174.068,41.486,158.071
C07992=1049.162,391.149,-124.237,174.075,41.492,158.073
C07993=1049.171,391.395,-124.279,174.083,41.499,158.075
C07994=1049.180,391.641,-124.322,174.090,41.505,158.077
C07995=1049.188,391.886,-124.364,174.096,41.511,158.078
C07996=1049.196,392.133,-124.406,174.104,41.518,158.081
C07997=1049.205,392.379,-124.449,174.111,41.524,158.083
C07998=1049.213,392.626,-124.491,174.118,41.530,158.084
C07999=1049.222,392.872,-124.534,174.126,41.537,158.087
C08000=1049.231,393.118,-124.576,174.133,41.543,158.089
C08001=1049.239,393.364,-124.619,174.139,41.550,158.091
C08002=1049.248,393.610,-124.662,174.147,41.556,158.093
C08003=1049.255,393.856,-124.705,174.154,41.562,158.095
C08004=1049.264,394.102,-124.747,174.161,41.569,158.097
C08005=1049.273,394.348,-124.790,174.169,41.575,158.099
C08006=1049.281,394.594,-124.833,174.176,41.582,158.101
C08007=1049.290,394.840,-124.876,174.184,41.588,158.103
C08008=1049.298,395.086,-124.919,174.191,41.595,158.105
C08009=1049.307,395.332,-124.962,174.198,41.601,158.107
C08010=1049.315,395.578,-125.005,174.206,41.608,158.109
C08011=1049.325,395.825,-125.048,174.213,41.614,158.111
C08012=1049.334,396.071,-125.091,174.221,41.621,158.113
C08013=1049.342,396.317,-125.134,174.228,41.627,158.115
C08014=1049.351,396.563,-125.177,174.236,41.634,158.117
C08015=1049.359,396.809,-125.220,174.243,41.641,158.120
C08016=1049.368,397.055,-125.263,174.251,41.647,158.122
C08017=1049.376,397.301,-125.306,174.258,41.654,158.124
C08018=1049.385,397.547,-125.349,174.266,41.661,158.126
C08019=1049.394,397.793,-125.393,174.273,41.668,158.128
C08020=1049.403,398.039,-125.436,174.281,41.674,158.130
C08021=1049.411,398.285,-125.479,174.288,41.681,158.132
C08022=1049.420,398.531,-125.523,174.296,41.687,158.135
C08023=1049.428,398.777,-125.566,174.303,41.695,158.137
C08024=1049.438,399.023,-125.610,174.311,41.701,158.139
C08025=1049.446,399.269,-125.653,174.319,41.708,158.141
C08026=1049.455,399.514,-125.697,174.326,41.715,158.143
C08027=1049.464,399.762,-125.741,174.334,41.722,158.146
C08028=1049.472,400.007,-125.784,174.341,41.729,158.148
C08029=1049.481,400.253,-125.827,174.349,41.736,158.150
C08030=1049.490,400.499,-125.871,174.358,41.742,158.152
C08031=1049.499,400.745,-125.914,174.365,41.749,158.154
C08032=1049.508,400.991,-125.959,174.373,41.756,158.157
C08033=1049.517,401.237,-126.002,174.380,41.763,158.159
C08034=1049.526,401.482,-126.046,174.388,41.770,158.161
C08035=1049.534,401.729,-126.090,174.397,41.777,158.163
C08036=1049.543,401.975,-126.134,174.405,41.784,158.166
C08037=1049.552,402.221,-126.178,174.412,41.791,158.168
C08038=1049.561,402.466,-126.222,174.420,41.798,158.170
C08039=1049.570,402.713,-126.266,174.428,41.806,158.173
C08040=1049.579,402.958,-126.310,174.436,41.813,158.175
C08041=1049.588,403.204,-126.354,174.444,41.820,158.177
C08042=1049.601,403.585,-126.422,174.456,41.831,158.181
C08043=1049.616,403.965,-126.491,174.469,41.842,158.184
C08044=1049.629,404.344,-126.559,174.481,41.853,158.188
C08045=1049.643,404.724,-126.628,174.494,41.864,158.192
C08046=1049.652,404.970,-126.672,174.502,41.872,158.194
C08047=1049.661,405.217,-126.717,174.510,41.879,158.196
C08048=1049.670,405.462,-126.761,174.519,41.886,158.199
C08049=1049.679,405.708,-126.806,174.527,41.894,158.201
C08050=1049.688,405.954,-126.851,174.536,41.901,158.204
C08051=1049.697,406.199,-126.895,174.544,41.908,158.206
C08052=1049.706,406.445,-126.940,174.552,41.916,158.209
C08053=1049.715,406.691,-126.984,174.560,41.923,158.211
C08054=1049.724,406.937,-127.030,174.568,41.931,158.213
C08055=1049.733,407.183,-127.074,174.577,41.938,158.216
C08056=1049.742,407.428,-127.119,174.585,41.946,158.218
C08057=1049.752,407.674,-127.164,174.594,41.953,158.221
C08058=1049.760,407.920,-127.209,174.602,41.961,158.223
C08059=1049.770,408.166,-127.253,174.611,41.968,158.226
C08060=1049.779,408.412,-127.299,174.619,41.976,158.228
C08061=1049.789,408.657,-127.344,174.628,41.983,158.231
C08062=1049.797,408.904,-127.388,174.636,41.991,158.233
C08063=1049.806,409.149,-127.434,174.645,41.998,158.236
C08064=1049.816,409.395,-127.479,174.653,42.006,158.238
C08065=1049.825,409.641,-127.524,174.662,42.014,158.241
C08066=1049.835,409.886,-127.569,174.671,42.021,158.243
C08067=1049.844,410.132,-127.614,174.679,42.029,158.246
C08068=1049.853,410.378,-127.659,174.688,42.037,158.248
C08069=1049.862,410.623,-127.704,174.697,42.045,158.251
C08070=1049.871,410.869,-127.750,174.706,42.052,158.253
C08071=1049.881,411.114,-127.795,174.715,42.060,158.256
C08072=1049.890,411.360,-127.841,174.723,42.068,158.259
C08073=1049.901,411.606,-127.886,174.732,42.076,158.261
C08074=1049.910,411.852,-127.931,174.741,42.084,158.264
C08075=1049.919,412.097,-127.978,174.750,42.091,158.266
C08076=1049.929,412.343,-128.022,174.758,42.099,158.269
C08077=1049.938,412.589,-128.068,174.768,42.107,158.272
C08078=1049.948,412.834,-128.114,174.777,42.115,158.274
C08079=1049.957,413.080,-128.159,174.786,42.123,158.277
C08080=1049.966,413.325,-128.205,174.795,42.131,158.280
C08081=1049.976,413.572,-128.251,174.804,42.139,158.282
C08082=1049.985,413.817,-128.297,174.813,42.147,158.285
C08083=1049.995,414.062,-128.343,174.822,42.155,158.288
C08084=1050.004,414.309,-128.389,174.831,42.163,158.291
C08085=1050.013,414.554,-128.435,174.841,42.171,158.293
C08086=1050.023,414.799,-128.481,174.850,42.180,158.296
C08087=1050.033,415.045,-128.528,174.858,42.188,158.299
C08088=1050.042,415.290,-128.574,174.868,42.196,158.302
C08089=1050.053,415.536,-128.620,174.877,42.204,158.304
C08090=1050.062,415.781,-128.666,174.887,42.213,158.307
C08091=1050.071,416.026,-128.712,174.896,42.221,158.310
C08092=1050.081,416.272,-128.759,174.905,42.229,158.313
C08093=1050.090,416.517,-128.805,174.915,42.237,158.316
C08094=1050.100,416.763,-128.851,174.924,42.246,158.318
C08095=1050.110,417.009,-128.898,174.934,42.254,158.321
C08096=1050.119,417.254,-128.944,174.943,42.263,158.324
C08097=1050.129,417.500,-128.990,174.953,42.271,158.327
C08098=1050.141,417.802,-129.048,174.965,42.281,158.330
C08099=1050.153,418.105,-129.106,174.976,42.292,158.334
C08100=1050.166,418.408,-129.163,174.989,42.302,158.338
C08101=1050.177,418.710,-129.220,175.000,42.313,158.341
C08102=1050.188,418.955,-129.267,175.011,42.321,158.344
C08103=1050.197,419.201,-129.314,175.020,42.330,158.347
C08104=1050.207,419.447,-129.362,175.030,42.338,158.350
C08105=1050.217,419.692,-129.408,175.040,42.347,158.353
C08106=1050.226,419.937,-129.455,175.049,42.355,158.356
C08107=1050.237,420.182,-129.502,175.060,42.364,158.359
C08108=1050.246,420.428,-129.550,175.070,42.373,158.362
C08109=1050.256,420.674,-129.597,175.079,42.381,158.365
C08110=1050.265,420.918,-129.643,175.089,42.390,158.368
C08111=1050.276,421.164,-129.691,175.100,42.399,158.371
C08112=1050.286,421.409,-129.738,175.109,42.408,158.374
C08113=1050.295,421.655,-129.786,175.119,42.417,158.377
C08114=1050.305,421.900,-129.833,175.130,42.426,158.380
C08115=1050.316,422.145,-129.880,175.140,42.435,158.383
C08116=1050.325,422.391,-129.928,175.149,42.443,158.386
C08117=1050.335,422.636,-129.975,175.160,42.452,158.389
C08118=1050.346,422.881,-130.023,175.170,42.462,158.392
C08119=1050.356,423.126,-130.070,175.181,42.470,158.395
C08120=1050.365,423.372,-130.118,175.191,42.479,158.398
C08121=1050.376,423.617,-130.165,175.202,42.488,158.402
C08122=1050.386,423.862,-130.213,175.211,42.497,158.405
C08123=1050.396,424.107,-130.260,175.222,42.506,158.408
C08124=1050.407,424.352,-130.309,175.232,42.515,158.411
C08125=1050.417,424.598,-130.357,175.243,42.525,158.414
C08126=1050.427,424.842,-130.404,175.253,42.534,158.417
C08127=1050.437,425.088,-130.452,175.264,42.543,158.421
C08128=1050.448,425.333,-130.501,175.274,42.552,158.424
C08129=1050.457,425.579,-130.548,175.285,42.561,158.427
C08130=1050.468,425.824,-130.596,175.296,42.571,158.430
C08131=1050.478,426.069,-130.645,175.306,42.580,158.434
C08132=1050.489,426.314,-130.693,175.318,42.589,158.437
C08133=1050.498,426.559,-130.742,175.329,42.599,158.440
C08134=1050.509,426.804,-130.790,175.339,42.608,158.443
C08135=1050.519,427.049,-130.838,175.350,42.618,158.447
C08136=1050.530,427.294,-130.886,175.361,42.627,158.450
C08137=1050.540,427.539,-130.935,175.372,42.637,158.453
C08138=1050.551,427.784,-130.983,175.382,42.646,158.457
C08139=1050.560,428.029,-131.032,175.394,42.656,158.460
C08140=1050.572,428.275,-131.080,175.405,42.665,158.464
C08141=1050.582,428.519,-131.129,175.416,42.674,158.467
C08142=1050.592,428.765,-131.178,175.427,42.684,158.470
C08143=1050.602,429.009,-131.226,175.439,42.694,158.474
C08144=1050.613,429.255,-131.275,175.450,42.703,158.477
C08145=1050.624,429.500,-131.324,175.461,42.713,158.481
C08146=1050.634,429.745,-131.373,175.473,42.723,158.484
C08147=1050.645,429.990,-131.422,175.484,42.732,158.487
C08148=1050.655,430.234,-131.471,175.495,42.743,158.491
C08149=1050.666,430.479,-131.520,175.507,42.752,158.494
C08150=1050.680,430.808,-131.587,175.522,42.766,158.499
C08151=1050.694,431.137,-131.653,175.537,42.779,158.504
C08152=1050.708,431.466,-131.718,175.553,42.792,158.509
C08153=1050.722,431.794,-131.785,175.569,42.806,158.514
C08154=1050.740,432.204,-131.868,175.588,42.823,158.520
C08155=1050.758,432.614,-131.951,175.608,42.839,158.526
C08156=1050.776,433.023,-132.033,175.628,42.856,158.532
C08157=1050.794,433.433,-132.117,175.648,42.874,158.538
C08158=1050.805,433.678,-132.166,175.659,42.884,158.542
C08159=1050.816,433.922,-132.216,175.671,42.894,158.545
C08160=1050.827,434.167,-132.266,175.684,42.904,158.549
C08161=1050.838,434.412,-132.316,175.695,42.914,158.553
C08162=1050.849,434.657,-132.365,175.708,42.925,158.557
C08163=1050.860,434.901,-132.416,175.720,42.935,158.560
C08164=1050.871,435.147,-132.466,175.732,42.945,158.564
C08165=1050.883,435.391,-132.516,175.745,42.956,158.568
C08166=1050.894,435.636,-132.566,175.757,42.966,158.572
C08167=1050.905,435.880,-132.616,175.769,42.977,158.576
C08168=1050.915,436.125,-132.666,175.781,42.987,158.579
C08169=1050.927,436.370,-132.716,175.794,42.998,158.583
C08170=1050.938,436.615,-132.767,175.807,43.008,158.587
C08171=1050.949,436.859,-132.817,175.819,43.019,158.591
C08172=1050.960,437.104,-132.867,175.832,43.030,158.595
C08173=1050.971,437.349,-132.918,175.844,43.040,158.599
C08174=1050.983,437.593,-132.969,175.857,43.051,158.603
C08175=1050.994,437.837,-133.019,175.870,43.062,158.607
C08176=1051.005,438.082,-133.070,175.882,43.072,158.611
C08177=1051.016,438.327,-133.121,175.896,43.083,158.615
C08178=1051.028,438.571,-133.172,175.909,43.094,158.619
C08179=1051.039,438.815,-133.222,175.922,43.105,158.623
C08180=1051.050,439.060,-133.274,175.935,43.116,158.627
C08181=1051.061,439.305,-133.325,175.947,43.127,158.631
C08182=1051.073,439.549,-133.376,175.961,43.138,158.635
C08183=1051.084,439.793,-133.427,175.974,43.149,158.639
C08184=1051.096,440.038,-133.478,175.987,43.160,158.643
C08185=1051.106,440.282,-133.529,176.001,43.171,158.647
C08186=1051.118,440.527,-133.581,176.014,43.182,158.651
C08187=1051.130,440.771,-133.632,176.027,43.193,158.656
C08188=1051.141,441.015,-133.683,176.041,43.205,158.660
C08189=1051.153,441.260,-133.735,176.054,43.216,158.664
C08190=1051.164,441.504,-133.787,176.068,43.227,158.668
C08191=1051.176,441.749,-133.838,176.081,43.239,158.673
C08192=1051.188,441.993,-133.889,176.096,43.250,158.677
C08193=1051.199,442.237,-133.942,176.109,43.261,158.681
C08194=1051.211,442.481,-133.993,176.123,43.272,158.685
C08195=1051.223,442.726,-134.045,176.136,43.284,158.690
C08196=1051.234,442.970,-134.097,176.150,43.295,158.694
C08197=1051.246,443.215,-134.149,176.165,43.307,158.699
C08198=1051.258,443.459,-134.201,176.178,43.319,158.703
C08199=1051.269,443.703,-134.252,176.192,43.330,158.707
C08200=1051.281,443.947,-134.305,176.207,43.341,158.712
C08201=1051.294,444.191,-134.357,176.220,43.353,158.716
C08202=1051.305,444.435,-134.410,176.234,43.365,158.721
C08203=1051.317,444.679,-134.462,176.249,43.377,158.725
C08204=1051.329,444.924,-134.514,176.263,43.389,158.730
C08205=1051.341,445.168,-134.566,176.278,43.400,158.734
C08206=1051.353,445.412,-134.618,176.292,43.412,158.739
C08207=1051.365,445.655,-134.672,176.307,43.424,158.743
C08208=1051.377,445.899,-134.724,176.322,43.435,158.748
C08209=1051.389,446.143,-134.776,176.336,43.448,158.752
C08210=1051.407,446.482,-134.848,176.356,43.464,158.759
C08211=1051.426,446.822,-134.919,176.377,43.480,158.765
C08212=1051.447,447.163,-134.990,176.398,43.496,158.771
C08213=1051.470,447.504,-135.060,176.419,43.511,158.777
C08214=1051.486,447.748,-135.109,176.434,43.522,158.782
C08215=1051.503,447.992,-135.157,176.449,43.533,158.786
C08216=1051.522,448.237,-135.205,176.464,43.543,158.790
C08217=1051.541,448.482,-135.252,176.480,43.554,158.795
C08218=1051.561,448.726,-135.299,176.495,43.564,158.799
C08219=1051.581,448.971,-135.345,176.510,43.574,158.803
C08220=1051.602,449.216,-135.391,176.526,43.584,158.807
C08221=1051.624,449.461,-135.436,176.542,43.594,158.811
C08222=1051.646,449.706,-135.481,176.557,43.604,158.815
C08223=1051.669,449.952,-135.525,176.574,43.613,158.819
C08224=1051.693,450.197,-135.569,176.589,43.622,158.823
C08225=1051.718,450.442,-135.612,176.605,43.632,158.827
C08226=1051.402,450.468,-135.909,176.605,43.727,158.855
C08227=1051.378,450.222,-135.866,176.588,43.717,158.851
C08228=1051.353,449.977,-135.823,176.572,43.708,158.847
C08229=1051.329,449.732,-135.779,176.557,43.699,158.843
C08230=1051.307,449.486,-135.733,176.541,43.689,158.839
C08231=1051.285,449.241,-135.688,176.525,43.679,158.834
C08232=1051.263,448.996,-135.644,176.510,43.669,158.830
C08233=1051.243,448.751,-135.597,176.494,43.659,158.826
C08234=1051.224,448.507,-135.550,176.479,43.649,158.822
C08235=1051.205,448.262,-135.503,176.463,43.639,158.818
C08236=1051.186,448.017,-135.455,176.448,43.629,158.813
C08237=1051.168,447.773,-135.406,176.432,43.618,158.809
C08238=1051.151,447.530,-135.358,176.417,43.607,158.805
C08239=1051.131,447.206,-135.292,176.397,43.593,158.799
C08240=1051.110,446.884,-135.226,176.377,43.578,158.793
C08241=1051.091,446.562,-135.158,176.358,43.563,158.787
C08242=1051.074,446.242,-135.091,176.339,43.547,158.781
C08243=1051.061,445.998,-135.039,176.324,43.536,158.776
C08244=1051.050,445.754,-134.986,176.309,43.524,158.772
C08245=1051.037,445.511,-134.933,176.295,43.512,158.767
C08246=1051.025,445.267,-134.881,176.280,43.501,158.763
C08247=1051.013,445.023,-134.829,176.266,43.489,158.758
C08248=1051.002,444.779,-134.776,176.251,43.477,158.754
C08249=1050.989,444.535,-134.724,176.237,43.465,158.749
C08250=1050.977,444.291,-134.672,176.222,43.454,158.745
C08251=1050.965,444.046,-134.619,176.208,43.442,158.740
C08252=1050.953,443.802,-134.567,176.193,43.431,158.736
C08253=1050.941,443.558,-134.515,176.180,43.419,158.731
C08254=1050.930,443.314,-134.463,176.165,43.408,158.727
C08255=1050.918,443.069,-134.411,176.151,43.396,158.723
C08256=1050.906,442.826,-134.359,176.138,43.385,158.718
C08257=1050.895,442.581,-134.307,176.124,43.373,158.714
C08258=1050.883,442.337,-134.255,176.109,43.362,158.710
C08259=1050.871,442.093,-134.204,176.096,43.351,158.705
C08260=1050.860,441.848,-134.152,176.082,43.339,158.701
C08261=1050.848,441.604,-134.101,176.069,43.328,158.697
C08262=1050.836,441.360,-134.048,176.055,43.317,158.692
C08263=1050.825,441.116,-133.997,176.042,43.306,158.688
C08264=1050.813,440.871,-133.945,176.027,43.294,158.684
C08265=1050.801,440.626,-133.894,176.014,43.284,158.680
C08266=1050.790,440.383,-133.843,176.000,43.272,158.676
C08267=1050.779,440.138,-133.792,175.987,43.262,158.672
C08268=1050.767,439.893,-133.741,175.974,43.250,158.667
C08269=1050.756,439.649,-133.689,175.960,43.239,158.663
C08270=1050.744,439.404,-133.638,175.948,43.228,158.659
C08271=1050.733,439.160,-133.587,175.935,43.218,158.655
C08272=1050.721,438.915,-133.536,175.922,43.207,158.651
C08273=1050.710,438.672,-133.485,175.908,43.196,158.647
C08274=1050.699,438.427,-133.434,175.895,43.185,158.643
C08275=1050.688,438.182,-133.383,175.882,43.174,158.639
C08276=1050.676,437.937,-133.332,175.870,43.163,158.635
C08277=1050.665,437.693,-133.282,175.857,43.153,158.631
C08278=1050.654,437.448,-133.231,175.844,43.142,158.627
C08279=1050.643,437.204,-133.180,175.831,43.132,158.623
C08280=1050.632,436.959,-133.130,175.818,43.121,158.619
C08281=1050.621,436.715,-133.079,175.805,43.110,158.615
C08282=1050.609,436.470,-133.029,175.792,43.100,158.611
C08283=1050.598,436.225,-132.978,175.781,43.089,158.607
C08284=1050.587,435.981,-132.928,175.768,43.079,158.604
C08285=1050.576,435.735,-132.878,175.756,43.068,158.600
C08286=1050.565,435.491,-132.828,175.743,43.058,158.596
C08287=1050.553,435.247,-132.778,175.731,43.047,158.592
C08288=1050.543,435.002,-132.728,175.718,43.038,158.588
C08289=1050.532,434.757,-132.678,175.706,43.027,158.585
C08290=1050.520,434.512,-132.627,175.693,43.017,158.581
C08291=1050.509,434.267,-132.578,175.682,43.006,158.577
C08292=1050.498,434.023,-132.527,175.669,42.997,158.573
C08293=1050.487,433.778,-132.478,175.657,42.986,158.569
C08294=1050.476,433.533,-132.428,175.645,42.976,158.566
C08295=1050.457,433.122,-132.344,175.624,42.959,158.560
C08296=1050.440,432.709,-132.261,175.605,42.942,158.553
C08297=1050.422,432.297,-132.178,175.585,42.925,158.547
C08298=1050.403,431.885,-132.094,175.565,42.908,158.541
C08299=1050.393,431.641,-132.045,175.554,42.898,158.538
C08300=1050.382,431.396,-131.995,175.542,42.888,158.534
C08301=1050.372,431.151,-131.946,175.531,42.879,158.531
C08302=1050.360,430.906,-131.897,175.518,42.869,158.527
C08303=1050.351,430.661,-131.848,175.507,42.859,158.523
C08304=1050.340,430.416,-131.799,175.495,42.849,158.520
C08305=1050.329,430.171,-131.749,175.484,42.839,158.516
C08306=1050.319,429.927,-131.700,175.472,42.830,158.513
C08307=1050.308,429.681,-131.652,175.461,42.820,158.509
C08308=1050.298,429.437,-131.602,175.449,42.810,158.506
C08309=1050.288,429.191,-131.553,175.438,42.801,158.502
C08310=1050.276,428.947,-131.504,175.427,42.791,158.499
C08311=1050.266,428.702,-131.456,175.415,42.781,158.496
C08312=1050.255,428.456,-131.408,175.405,42.771,158.492
C08313=1050.245,428.212,-131.358,175.394,42.762,158.489
C08314=1050.235,427.966,-131.309,175.383,42.753,158.485
C08315=1050.224,427.722,-131.262,175.371,42.743,158.482
C08316=1050.214,427.476,-131.213,175.360,42.734,158.479
C08317=1050.204,427.231,-131.165,175.349,42.725,158.475
C08318=1050.193,426.986,-131.116,175.339,42.715,158.472
C08319=1050.183,426.741,-131.068,175.328,42.706,158.469
C08320=1050.173,426.496,-131.019,175.316,42.696,158.465
C08321=1050.162,426.251,-130.971,175.305,42.687,158.462
C08322=1050.152,426.006,-130.923,175.295,42.678,158.459
C08323=1050.142,425.761,-130.875,175.284,42.668,158.456
C08324=1050.132,425.516,-130.826,175.273,42.659,158.452
C08325=1050.121,425.271,-130.778,175.263,42.650,158.449
C08326=1050.111,425.025,-130.730,175.252,42.641,158.446
C08327=1050.101,424.780,-130.682,175.241,42.632,158.443
C08328=1050.091,424.535,-130.635,175.231,42.622,158.439
C08329=1050.079,424.290,-130.587,175.220,42.614,158.436
C08330=1050.070,424.044,-130.539,175.210,42.604,158.433
C08331=1050.060,423.824,-130.495,175.201,42.597,158.430
C08332=1050.052,423.605,-130.453,175.191,42.588,158.427
C08333=1050.042,423.384,-130.411,175.182,42.581,158.425
C08334=1050.033,423.165,-130.368,175.172,42.572,158.422
C08335=1050.024,422.944,-130.324,175.163,42.565,158.419
C08336=1050.015,422.724,-130.282,175.154,42.556,158.416
C08337=1050.006,422.504,-130.240,175.145,42.548,158.413
C08338=1049.997,422.284,-130.197,175.135,42.540,158.411
C08339=1049.987,422.039,-130.149,175.125,42.532,158.408
C08340=1049.977,421.793,-130.102,175.115,42.523,158.405
C08341=1049.967,421.548,-130.054,175.105,42.514,158.402
C08342=1049.957,421.303,-130.007,175.095,42.505,158.399
C08343=1049.946,421.058,-129.960,175.084,42.496,158.395
C08344=1049.937,420.812,-129.912,175.074,42.488,158.392
C08345=1049.928,420.567,-129.866,175.065,42.479,158.390
C08346=1049.918,420.321,-129.819,175.054,42.470,158.386
C08347=1049.907,420.076,-129.772,175.044,42.462,158.383
C08348=1049.898,419.831,-129.724,175.035,42.453,158.381
C08349=1049.888,419.585,-129.677,175.025,42.444,158.377
C08350=1049.878,419.340,-129.630,175.014,42.436,158.375
C08351=1049.870,419.120,-129.588,175.006,42.428,158.372
C08352=1049.861,418.901,-129.546,174.997,42.421,158.369
C08353=1049.852,418.681,-129.505,174.989,42.413,158.367
C08354=1049.843,418.462,-129.462,174.979,42.405,158.364
C08355=1049.834,418.242,-129.420,174.971,42.398,158.362
C08356=1049.825,418.022,-129.379,174.962,42.391,158.359
C08357=1049.816,417.803,-129.337,174.954,42.383,158.356
C08358=1049.808,417.583,-129.295,174.945,42.375,158.354
C08359=1049.798,417.338,-129.249,174.935,42.367,158.351
C08360=1049.789,417.092,-129.202,174.926,42.359,158.348
C08361=1049.779,416.847,-129.156,174.916,42.351,158.345
C08362=1049.768,416.602,-129.110,174.907,42.342,158.342
C08363=1049.758,416.356,-129.063,174.897,42.334,158.340
C08364=1049.749,416.111,-129.017,174.888,42.325,158.337
C08365=1049.739,415.865,-128.971,174.878,42.318,158.334
C08366=1049.730,415.619,-128.924,174.869,42.309,158.331
C08367=1049.720,415.374,-128.878,174.860,42.301,158.329
C08368=1049.711,415.128,-128.832,174.850,42.293,158.326
C08369=1049.702,414.883,-128.786,174.841,42.285,158.323
C08370=1049.692,414.637,-128.740,174.832,42.277,158.320
C08371=1049.683,414.391,-128.694,174.823,42.268,158.317
C08372=1049.673,414.145,-128.647,174.814,42.260,158.315
C08373=1049.664,413.900,-128.601,174.805,42.253,158.312
C08374=1049.655,413.654,-128.556,174.795,42.245,158.309
C08375=1049.645,413.410,-128.510,174.786,42.236,158.307
C08376=1049.635,413.164,-128.464,174.777,42.228,158.304
C08377=1049.626,412.918,-128.418,174.768,42.220,158.301
C08378=1049.616,412.673,-128.372,174.759,42.213,158.299
C08379=1049.607,412.426,-128.326,174.750,42.205,158.296
C08380=1049.597,412.181,-128.281,174.741,42.197,158.293
C08381=1049.588,411.935,-128.235,174.731,42.189,158.291
C08382=1049.578,411.690,-128.191,174.723,42.181,158.288
C08383=1049.569,411.443,-128.145,174.714,42.174,158.285
C08384=1049.559,411.198,-128.099,174.705,42.166,158.283
C08385=1049.550,410.953,-128.054,174.696,42.158,158.280
C08386=1049.541,410.707,-128.008,174.688,42.150,158.278
C08387=1049.531,410.461,-127.964,174.679,42.143,158.275
C08388=1049.522,410.215,-127.918,174.670,42.135,158.273
C08389=1049.512,409.970,-127.873,174.661,42.127,158.270
C08390=1049.503,409.724,-127.828,174.652,42.120,158.267
C08391=1049.494,409.478,-127.782,174.643,42.112,158.265
C08392=1049.484,409.232,-127.737,174.635,42.105,158.262
C08393=1049.475,408.986,-127.692,174.626,42.097,158.260
C08394=1049.465,408.741,-127.647,174.618,42.089,158.257
C08395=1049.457,408.496,-127.602,174.609,42.082,158.255
C08396=1049.447,408.250,-127.557,174.601,42.074,158.252
C08397=1049.438,408.004,-127.512,174.592,42.067,158.250
C08398=1049.429,407.758,-127.468,174.584,42.059,158.247
C08399=1049.420,407.512,-127.422,174.575,42.052,158.245
C08400=1049.411,407.266,-127.377,174.567,42.044,158.242
C08401=1049.401,407.020,-127.333,174.558,42.037,158.240
C08402=1049.392,406.775,-127.287,174.550,42.030,158.238
C08403=1049.383,406.530,-127.243,174.541,42.022,158.235
C08404=1049.375,406.283,-127.198,174.533,42.014,158.233
C08405=1049.365,406.038,-127.153,174.524,42.008,158.230
C08406=1049.356,405.791,-127.109,174.516,42.000,158.228
C08407=1049.347,405.547,-127.064,174.509,41.993,158.226
C08408=1049.338,405.300,-127.019,174.500,41.985,158.223
C08409=1049.329,405.054,-126.975,174.492,41.978,158.221
C08410=1049.321,404.809,-126.930,174.483,41.971,158.218
C08411=1049.306,404.427,-126.861,174.471,41.960,158.215
C08412=1049.292,404.044,-126.792,174.458,41.949,158.211
C08413=1049.279,403.662,-126.724,174.446,41.938,158.207
C08414=1049.264,403.280,-126.655,174.433,41.927,158.204
C08415=1049.255,403.034,-126.611,174.425,41.919,158.201
C08416=1049.246,402.788,-126.567,174.417,41.912,158.199
C08417=1049.238,402.543,-126.523,174.408,41.905,158.197
C08418=1049.229,402.296,-126.478,174.401,41.898,158.194
C08419=1049.220,402.051,-126.435,174.393,41.891,158.192
C08420=1049.210,401.805,-126.391,174.385,41.884,158.190
C08421=1049.202,401.559,-126.346,174.377,41.877,158.188
C08422=1049.193,401.312,-126.303,174.369,41.870,158.185
C08423=1049.184,401.067,-126.259,174.361,41.864,158.183
C08424=1049.175,400.821,-126.215,174.353,41.856,158.181
C08425=1049.166,400.575,-126.171,174.346,41.849,158.179
C08426=1049.158,400.329,-126.128,174.338,41.843,158.176
C08427=1049.148,400.083,-126.084,174.329,41.836,158.174
C08428=1049.140,399.837,-126.041,174.322,41.829,158.172
C08429=1049.130,399.591,-125.997,174.314,41.822,158.170
C08430=1049.122,399.345,-125.954,174.306,41.815,158.168
C08431=1049.114,399.099,-125.910,174.299,41.808,158.165
C08432=1049.105,398.853,-125.867,174.291,41.802,158.163
C08433=1049.096,398.607,-125.823,174.284,41.795,158.161
C08434=1049.087,398.361,-125.779,174.276,41.789,158.159
C08435=1049.079,398.115,-125.736,174.267,41.782,158.157
C08436=1049.070,397.869,-125.693,174.260,41.775,158.154
C08437=1049.061,397.623,-125.649,174.252,41.768,158.152
C08438=1049.052,397.377,-125.606,174.245,41.762,158.150
C08439=1049.044,397.131,-125.563,174.237,41.755,158.148
C08440=1049.035,396.885,-125.520,174.230,41.749,158.146
C08441=1049.027,396.639,-125.477,174.222,41.742,158.144
C08442=1049.018,396.393,-125.433,174.215,41.735,158.142
C08443=1049.010,396.147,-125.390,174.207,41.729,158.140
C08444=1049.001,395.900,-125.347,174.200,41.722,158.138
C08445=1048.991,395.654,-125.305,174.192,41.716,158.135
C08446=1048.983,395.408,-125.262,174.185,41.709,158.133
C08447=1048.974,395.162,-125.219,174.177,41.702,158.131
C08448=1048.966,394.916,-125.176,174.170,41.696,158.129
C08449=1048.957,394.670,-125.133,174.163,41.690,158.127
C08450=1048.949,394.424,-125.089,174.155,41.683,158.125
C08451=1048.940,394.178,-125.047,174.149,41.677,158.123
C08452=1048.931,393.932,-125.004,174.141,41.670,158.121
C08453=1048.923,393.686,-124.962,174.134,41.664,158.119
C08454=1048.914,393.440,-124.919,174.127,41.658,158.117
C08455=1048.906,393.194,-124.876,174.119,41.651,158.115
C08456=1048.897,392.948,-124.833,174.112,41.645,158.113
C08457=1048.889,392.702,-124.791,174.105,41.639,158.111
C08458=1048.881,392.456,-124.748,174.097,41.632,158.109
C08459=1048.872,392.210,-124.705,174.091,41.626,158.107
C08460=1048.863,391.963,-124.664,174.084,41.620,158.105
C08461=1048.855,391.717,-124.620,174.076,41.613,158.103
C08462=1048.846,391.471,-124.578,174.069,41.607,158.101
C08463=1048.837,391.224,-124.536,174.062,41.601,158.099
C08464=1048.830,390.979,-124.494,174.054,41.595,158.097
C08465=1048.821,390.732,-124.451,174.048,41.589,158.095
C08466=1048.812,390.487,-124.409,174.041,41.583,158.093
C08467=1048.800,390.123,-124.347,174.030,41.573,158.090
C08468=1048.788,389.759,-124.284,174.020,41.564,158.087
C08469=1048.775,389.396,-124.222,174.010,41.555,158.084
C08470=1048.763,389.033,-124.160,173.999,41.546,158.082
C08471=1048.754,388.787,-124.118,173.992,41.540,158.080
C08472=1048.746,388.540,-124.076,173.985,41.534,158.078
C08473=1048.737,388.294,-124.034,173.979,41.528,158.076
C08474=1048.729,388.048,-123.993,173.972,41.522,158.074
C08475=1048.721,387.801,-123.951,173.964,41.516,158.072
C08476=1048.712,387.555,-123.909,173.958,41.510,158.070
C08477=1048.704,387.309,-123.868,173.951,41.504,158.068
C08478=1048.695,387.063,-123.825,173.944,41.499,158.067
C08479=1048.687,386.816,-123.784,173.938,41.492,158.065
C08480=1048.679,386.570,-123.742,173.931,41.487,158.063
C08481=1048.670,386.323,-123.701,173.923,41.481,158.061
C08482=1048.662,386.078,-123.659,173.917,41.475,158.059
C08483=1048.654,385.830,-123.618,173.910,41.469,158.057
C08484=1048.646,385.585,-123.576,173.903,41.463,158.055
C08485=1048.637,385.338,-123.535,173.897,41.458,158.054
C08486=1048.629,385.092,-123.493,173.890,41.451,158.052
C08487=1048.620,384.845,-123.452,173.884,41.446,158.050
C08488=1048.612,384.600,-123.410,173.877,41.440,158.048
C08489=1048.604,384.352,-123.369,173.869,41.434,158.046
C08490=1048.596,384.107,-123.327,173.863,41.428,158.044
C08491=1048.587,383.860,-123.286,173.856,41.423,158.043
C08492=1048.580,383.614,-123.244,173.850,41.417,158.041
C08493=1048.572,383.367,-123.204,173.843,41.411,158.039
C08494=1048.563,383.121,-123.162,173.837,41.406,158.037
C08495=1048.555,382.875,-123.121,173.830,41.400,158.036
C08496=1048.547,382.628,-123.079,173.824,41.394,158.034
C08497=1048.538,382.382,-123.039,173.817,41.388,158.032
C08498=1048.531,382.135,-122.997,173.811,41.382,158.030
C08499=1048.522,381.889,-122.956,173.804,41.377,158.028
C08500=1048.514,381.643,-122.915,173.798,41.371,158.027
C08501=1048.506,381.396,-122.874,173.791,41.366,158.025
C08502=1048.499,381.150,-122.833,173.785,41.360,158.023
C08503=1048.490,380.903,-122.792,173.778,41.355,158.022
C08504=1048.482,380.657,-122.751,173.772,41.349,158.020
C08505=1048.475,380.411,-122.710,173.766,41.343,158.018
C08506=1048.467,380.164,-122.669,173.759,41.338,158.016
C08507=1048.459,379.918,-122.628,173.753,41.332,158.015
C08508=1048.450,379.671,-122.587,173.746,41.327,158.013
C08509=1048.443,379.424,-122.546,173.740,41.321,158.011
C08510=1048.434,379.178,-122.506,173.734,41.316,158.010
C08511=1048.426,378.932,-122.465,173.727,41.310,158.008
C08512=1048.417,378.685,-122.424,173.721,41.305,158.006
C08513=1048.410,378.438,-122.384,173.714,41.299,158.004
C08514=1048.402,378.192,-122.344,173.709,41.294,158.003
C08515=1048.394,377.946,-122.303,173.703,41.289,158.001
C08516=1048.386,377.699,-122.263,173.696,41.283,158.000
C08517=1048.377,377.453,-122.222,173.690,41.278,157.998
C08518=1048.370,377.206,-122.182,173.684,41.272,157.996
C08519=1048.361,376.959,-122.141,173.677,41.267,157.995
C08520=1048.353,376.713,-122.100,173.671,41.262,157.993
C08521=1048.345,376.466,-122.060,173.665,41.256,157.991
C08522=1048.337,376.220,-122.020,173.659,41.251,157.990
C08523=1048.327,375.889,-121.966,173.651,41.244,157.987
C08524=1048.316,375.559,-121.912,173.643,41.237,157.985
C08525=1048.306,375.228,-121.858,173.634,41.230,157.983
C08526=1048.295,374.898,-121.804,173.626,41.223,157.981
C08527=1048.287,374.651,-121.764,173.620,41.218,157.979
C08528=1048.279,374.405,-121.724,173.614,41.212,157.978
C08529=1048.271,374.158,-121.684,173.608,41.207,157.976
C08530=1048.264,373.911,-121.644,173.601,41.202,157.975
C08531=1048.256,373.665,-121.603,173.596,41.197,157.973
C08532=1048.248,373.418,-121.563,173.590,41.192,157.971
C08533=1048.240,373.171,-121.523,173.584,41.186,157.970
C08534=1048.232,372.925,-121.483,173.577,41.181,157.968
C08535=1048.225,372.679,-121.443,173.571,41.176,157.967
C08536=1048.217,372.432,-121.404,173.566,41.171,157.965
C08537=1048.209,372.185,-121.364,173.560,41.166,157.964
C08538=1048.201,371.938,-121.324,173.554,41.161,157.962
C08539=1048.193,371.692,-121.284,173.549,41.156,157.961
C08540=1048.185,371.445,-121.244,173.542,41.151,157.959
C08541=1048.178,371.199,-121.204,173.536,41.146,157.957
C08542=1048.170,370.952,-121.165,173.530,41.140,157.956
C08543=1048.162,370.705,-121.125,173.525,41.136,157.954
C08544=1048.154,370.458,-121.085,173.519,41.130,157.953
C08545=1048.146,370.212,-121.046,173.513,41.126,157.951
C08546=1048.139,369.965,-121.007,173.507,41.120,157.950
C08547=1048.131,369.718,-120.967,173.501,41.116,157.948
C08548=1048.123,369.472,-120.927,173.495,41.111,157.947
C08549=1048.115,369.225,-120.888,173.489,41.106,157.945
C08550=1048.107,368.978,-120.848,173.484,41.101,157.944
C08551=1048.100,368.731,-120.809,173.478,41.096,157.942
C08552=1048.092,368.485,-120.770,173.472,41.091,157.941
C08553=1048.084,368.238,-120.730,173.467,41.086,157.939
C08554=1048.076,367.992,-120.691,173.461,41.081,157.938
C08555=1048.069,367.744,-120.652,173.455,41.076,157.936
C08556=1048.061,367.497,-120.612,173.450,41.072,157.935
C08557=1048.053,367.252,-120.573,173.443,41.066,157.933
C08558=1048.046,367.004,-120.534,173.437,41.062,157.932
C08559=1048.037,366.757,-120.495,173.432,41.057,157.931
C08560=1048.030,366.511,-120.456,173.426,41.052,157.929
C08561=1048.022,366.264,-120.416,173.420,41.047,157.928
C08562=1048.015,366.017,-120.378,173.415,41.042,157.926
C08563=1048.007,365.771,-120.338,173.409,41.038,157.925
C08564=1047.999,365.523,-120.299,173.404,41.033,157.923
C08565=1047.992,365.277,-120.259,173.398,41.028,157.922
C08566=1047.984,365.030,-120.221,173.392,41.023,157.920
C08567=1047.977,364.783,-120.182,173.387,41.018,157.919
C08568=1047.969,364.536,-120.143,173.381,41.014,157.917
C08569=1047.962,364.289,-120.104,173.376,41.009,157.916
C08570=1047.954,364.042,-120.065,173.370,41.004,157.915
C08571=1047.947,363.796,-120.026,173.364,41.000,157.913
C08572=1047.938,363.549,-119.987,173.360,40.995,157.912
C08573=1047.932,363.302,-119.948,173.354,40.990,157.910
C08574=1047.924,363.055,-119.910,173.349,40.985,157.909
C08575=1047.916,362.808,-119.870,173.343,40.981,157.908
C08576=1047.909,362.562,-119.832,173.338,40.976,157.906
C08577=1047.901,362.315,-119.793,173.332,40.971,157.905
C08578=1047.894,362.068,-119.754,173.326,40.967,157.903
C08579=1047.884,361.756,-119.706,173.319,40.961,157.902
C08580=1047.874,361.445,-119.657,173.313,40.955,157.900
C08581=1047.864,361.134,-119.609,173.306,40.949,157.898
C08582=1047.855,360.822,-119.561,173.299,40.944,157.896
C08583=1047.847,360.576,-119.522,173.293,40.939,157.895
C08584=1047.839,360.328,-119.484,173.288,40.935,157.894
C08585=1047.832,360.082,-119.445,173.283,40.930,157.892
C08586=1047.825,359.835,-119.407,173.278,40.925,157.891
C08587=1047.817,359.588,-119.368,173.272,40.921,157.890
C08588=1047.809,359.341,-119.330,173.267,40.916,157.888
C08589=1047.802,359.094,-119.292,173.261,40.912,157.887
C08590=1047.795,358.847,-119.253,173.256,40.907,157.886
C08591=1047.787,358.600,-119.215,173.250,40.903,157.884
C08592=1047.779,358.354,-119.177,173.246,40.898,157.883
C08593=1047.772,358.107,-119.139,173.240,40.894,157.882
C08594=1047.764,357.859,-119.100,173.235,40.889,157.880
C08595=1047.757,357.613,-119.062,173.230,40.885,157.879
C08596=1047.750,357.365,-119.024,173.224,40.881,157.878
C08597=1047.742,357.119,-118.986,173.220,40.876,157.876
C08598=1047.735,356.871,-118.948,173.214,40.872,157.875
C08599=1047.727,356.625,-118.910,173.209,40.867,157.874
C08600=1047.720,356.377,-118.872,173.203,40.863,157.873
C08601=1047.712,356.131,-118.834,173.198,40.859,157.871
C08602=1047.705,355.884,-118.796,173.193,40.854,157.870
C08603=1047.697,355.637,-118.758,173.188,40.850,157.869
C08604=1047.690,355.389,-118.720,173.183,40.846,157.867
C08605=1047.682,355.142,-118.683,173.177,40.841,157.866
C08606=1047.675,354.896,-118.644,173.172,40.837,157.865
C08607=1047.668,354.649,-118.607,173.167,40.833,157.864
C08608=1047.660,354.402,-118.569,173.162,40.829,157.862
C08609=1047.652,354.154,-118.531,173.157,40.824,157.861
C08610=1047.645,353.907,-118.493,173.152,40.819,157.860
C08611=1047.638,353.660,-118.456,173.147,40.815,157.858
C08612=1047.630,353.413,-118.417,173.141,40.811,157.857
C08613=1047.623,353.166,-118.380,173.136,40.807,157.856
C08614=1047.616,352.919,-118.342,173.132,40.803,157.855
C08615=1047.608,352.672,-118.305,173.126,40.798,157.853
C08616=1047.601,352.425,-118.267,173.121,40.794,157.852
C08617=1047.594,352.178,-118.230,173.117,40.790,157.851
C08618=1047.586,351.932,-118.192,173.111,40.786,157.850
C08619=1047.578,351.684,-118.155,173.106,40.782,157.848
C08620=1047.571,351.437,-118.117,173.101,40.777,157.847
C08621=1047.564,351.190,-118.080,173.096,40.773,157.846
C08622=1047.557,350.943,-118.042,173.091,40.769,157.845
C08623=1047.549,350.696,-118.005,173.086,40.765,157.843
C08624=1047.542,350.449,-117.967,173.081,40.760,157.842
C08625=1047.535,350.202,-117.929,173.076,40.756,157.841
C08626=1047.527,349.954,-117.893,173.071,40.752,157.840
C08627=1047.520,349.707,-117.856,173.066,40.748,157.839
C08628=1047.513,349.460,-117.818,173.061,40.744,157.837
C08629=1047.506,349.213,-117.781,173.056,40.740,157.836
C08630=1047.498,348.966,-117.744,173.051,40.736,157.835
C08631=1047.490,348.719,-117.706,173.047,40.731,157.834
C08632=1047.483,348.471,-117.669,173.042,40.728,157.833
C08633=1047.476,348.225,-117.633,173.036,40.724,157.831
C08634=1047.469,347.978,-117.595,173.032,40.719,157.830
C08635=1047.460,347.672,-117.550,173.025,40.715,157.829
C08636=1047.450,347.366,-117.504,173.020,40.709,157.827
C08637=1047.442,347.060,-117.457,173.013,40.705,157.826
C08638=1047.433,346.754,-117.412,173.007,40.699,157.824
C08639=1047.425,346.507,-117.375,173.002,40.696,157.823
C08640=1047.418,346.260,-117.338,172.998,40.691,157.822
C08641=1047.411,346.013,-117.301,172.993,40.688,157.821
C08642=1047.403,345.766,-117.264,172.988,40.683,157.820
C08643=1047.396,345.518,-117.227,172.983,40.679,157.818
C08644=1047.389,345.271,-117.190,172.979,40.675,157.817
C08645=1047.382,345.024,-117.154,172.974,40.671,157.816
C08646=1047.375,344.777,-117.117,172.969,40.667,157.815
C08647=1047.367,344.530,-117.080,172.964,40.663,157.814
C08648=1047.360,344.282,-117.043,172.960,40.659,157.813
C08649=1047.354,344.035,-117.006,172.955,40.656,157.812
C08650=1047.346,343.788,-116.970,172.950,40.651,157.810
C08651=1047.339,343.540,-116.933,172.945,40.648,157.809
C08652=1047.332,343.294,-116.897,172.941,40.643,157.808
C08653=1047.325,343.046,-116.860,172.936,40.640,157.807
C08654=1047.317,342.799,-116.824,172.932,40.636,157.806
C08655=1047.310,342.552,-116.786,172.926,40.632,157.805
C08656=1047.303,342.305,-116.750,172.922,40.628,157.804
C08657=1047.296,342.057,-116.714,172.917,40.625,157.803
C08658=1047.288,341.810,-116.677,172.913,40.620,157.801
C08659=1047.282,341.563,-116.641,172.907,40.617,157.800
C08660=1047.274,341.315,-116.605,172.903,40.613,157.799
C08661=1047.266,341.068,-116.568,172.898,40.609,157.798
C08662=1047.260,340.821,-116.532,172.894,40.605,157.797
C08663=1047.252,340.574,-116.495,172.889,40.601,157.796
C08664=1047.245,340.327,-116.459,172.884,40.597,157.795
C08665=1047.238,340.080,-116.422,172.880,40.594,157.794
C08666=1047.230,339.832,-116.386,172.875,40.590,157.793
C08667=1047.223,339.585,-116.350,172.871,40.586,157.792
C08668=1047.216,339.338,-116.314,172.866,40.583,157.790
C08669=1047.210,339.090,-116.278,172.861,40.578,157.789
C08670=1047.202,338.843,-116.242,172.856,40.575,157.788
C08671=1047.196,338.596,-116.206,172.852,40.571,157.787
C08672=1047.188,338.348,-116.169,172.848,40.567,157.786
C08673=1047.180,338.101,-116.133,172.843,40.563,157.785
C08674=1047.174,337.854,-116.097,172.839,40.560,157.784
C08675=1047.166,337.606,-116.061,172.834,40.556,157.783
C08676=1047.159,337.359,-116.025,172.829,40.552,157.782
C08677=1047.152,337.111,-115.989,172.825,40.548,157.781
C08678=1047.145,336.864,-115.953,172.820,40.545,157.780
C08679=1047.138,336.618,-115.917,172.816,40.541,157.778
C08680=1047.131,336.370,-115.881,172.812,40.537,157.777
C08681=1047.125,336.123,-115.845,172.807,40.534,157.776
C08682=1047.117,335.875,-115.809,172.802,40.530,157.775
C08683=1047.110,335.628,-115.774,172.798,40.526,157.774
C08684=1047.102,335.380,-115.737,172.793,40.522,157.773
C08685=1047.095,335.134,-115.702,172.789,40.519,157.772
C08686=1047.088,334.886,-115.666,172.785,40.515,157.771
C08687=1047.081,334.639,-115.630,172.780,40.512,157.770
C08688=1047.074,334.391,-115.595,172.776,40.508,157.769
C08689=1047.067,334.144,-115.559,172.772,40.504,157.768
C08690=1047.060,333.897,-115.524,172.767,40.501,157.767
C08691=1047.051,333.587,-115.479,172.761,40.496,157.766
C08692=1047.042,333.277,-115.434,172.756,40.492,157.764
C08693=1047.034,332.968,-115.390,172.750,40.487,157.763
C08694=1047.024,332.659,-115.345,172.745,40.483,157.762
C08695=1047.017,332.411,-115.309,172.740,40.479,157.761
C08696=1047.010,332.163,-115.274,172.736,40.476,157.760
C08697=1047.003,331.916,-115.238,172.732,40.472,157.759
C08698=1046.996,331.668,-115.202,172.728,40.468,157.758
C08699=1046.990,331.421,-115.167,172.723,40.465,157.757
C08700=1046.983,331.174,-115.131,172.719,40.462,157.756
C08701=1046.976,330.927,-115.096,172.714,40.458,157.755
C08702=1046.968,330.678,-115.061,172.710,40.455,157.754
C08703=1046.962,330.431,-115.026,172.705,40.451,157.753
C08704=1046.955,330.184,-114.990,172.701,40.447,157.752
C08705=1046.948,329.937,-114.955,172.697,40.444,157.751
C08706=1046.940,329.689,-114.919,172.693,40.440,157.750
C08707=1046.934,329.442,-114.884,172.688,40.437,157.749
C08708=1046.926,329.195,-114.849,172.684,40.433,157.748
C08709=1046.919,328.946,-114.814,172.680,40.430,157.747
C08710=1046.912,328.699,-114.779,172.676,40.426,157.746
C08711=1046.905,328.452,-114.744,172.671,40.423,157.745
C08712=1046.898,328.205,-114.709,172.667,40.420,157.744
C08713=1046.890,327.957,-114.674,172.663,40.416,157.743
C08714=1046.883,327.710,-114.639,172.659,40.413,157.742
C08715=1046.876,327.462,-114.604,172.655,40.410,157.741
C08716=1046.869,327.215,-114.569,172.650,40.406,157.740
C08717=1046.861,326.967,-114.534,172.646,40.403,157.739
C08718=1046.854,326.720,-114.499,172.642,40.399,157.738
C08719=1046.847,326.472,-114.465,172.638,40.396,157.737
C08720=1046.840,326.225,-114.430,172.633,40.393,157.736
C08721=1046.833,325.978,-114.395,172.629,40.389,157.735
C08722=1046.826,325.730,-114.360,172.625,40.386,157.734
C08723=1046.819,325.482,-114.325,172.621,40.382,157.733
C08724=1046.812,325.235,-114.291,172.617,40.379,157.732
C08725=1046.805,324.987,-114.256,172.613,40.376,157.731
C08726=1046.797,324.740,-114.221,172.608,40.372,157.730
C08727=1046.791,324.493,-114.186,172.604,40.369,157.729
C08728=1046.784,324.245,-114.152,172.600,40.366,157.728
C08729=1046.777,323.998,-114.117,172.596,40.363,157.728
C08730=1046.770,323.750,-114.082,172.592,40.359,157.726
C08731=1046.763,323.503,-114.048,172.588,40.355,157.726
C08732=1046.756,323.255,-114.013,172.584,40.352,157.725
C08733=1046.749,323.008,-113.978,172.579,40.349,157.724
C08734=1046.742,322.760,-113.944,172.575,40.346,157.723
C08735=1046.735,322.513,-113.909,172.571,40.343,157.722
C08736=1046.728,322.265,-113.875,172.567,40.339,157.721
C08737=1046.721,322.018,-113.840,172.563,40.336,157.720
C08738=1046.714,321.771,-113.805,172.559,40.332,157.719
C08739=1046.707,321.523,-113.771,172.555,40.329,157.718
C08740=1046.700,321.275,-113.736,172.551,40.326,157.717
C08741=1046.693,321.028,-113.702,172.547,40.323,157.716
C08742=1046.686,320.780,-113.667,172.543,40.320,157.715
C08743=1046.679,320.533,-113.633,172.538,40.316,157.715
C08744=1046.673,320.285,-113.599,172.534,40.313,157.713
C08745=1046.665,320.038,-113.564,172.530,40.309,157.713
C08746=1046.659,319.790,-113.530,172.526,40.306,157.712
C08747=1046.650,319.475,-113.486,172.521,40.302,157.711
C08748=1046.642,319.161,-113.442,172.517,40.298,157.709
C08749=1046.632,318.847,-113.399,172.511,40.294,157.708
C08750=1046.623,318.531,-113.355,172.506,40.290,157.707
C08751=1046.617,318.284,-113.320,172.502,40.287,157.706
C08752=1046.610,318.037,-113.287,172.498,40.283,157.705
C08753=1046.604,317.789,-113.252,172.494,40.280,157.704
C08754=1046.596,317.541,-113.218,172.490,40.276,157.703
C08755=1046.590,317.294,-113.183,172.486,40.273,157.702
C08756=1046.583,317.047,-113.150,172.482,40.270,157.702
C08757=1046.577,316.799,-113.115,172.479,40.267,157.701
C08758=1046.569,316.551,-113.081,172.475,40.264,157.700
C08759=1046.563,316.303,-113.047,172.471,40.261,157.699
C08760=1046.555,316.056,-113.013,172.467,40.258,157.698
C08761=1046.550,315.809,-112.978,172.463,40.254,157.697
C08762=1046.542,315.561,-112.945,172.459,40.251,157.696
C08763=1046.536,315.313,-112.910,172.455,40.248,157.695
C08764=1046.529,315.066,-112.877,172.451,40.245,157.694
C08765=1046.523,314.818,-112.842,172.447,40.241,157.694
C08766=1046.516,314.571,-112.809,172.443,40.238,157.693
C08767=1046.509,314.323,-112.774,172.439,40.235,157.692
C08768=1046.503,314.076,-112.741,172.435,40.232,157.691
C08769=1046.496,313.828,-112.706,172.431,40.228,157.690
C08770=1046.489,313.581,-112.672,172.427,40.225,157.689
C08771=1046.483,313.333,-112.638,172.423,40.222,157.688
C08772=1046.476,313.085,-112.605,172.420,40.219,157.687
C08773=1046.470,312.838,-112.570,172.416,40.216,157.686
C08774=1046.463,312.590,-112.537,172.412,40.213,157.686
C08775=1046.456,312.342,-112.503,172.409,40.209,157.685
C08776=1046.448,312.095,-112.469,172.405,40.207,157.684
C08777=1046.442,311.848,-112.436,172.401,40.203,157.683
C08778=1046.435,311.599,-112.402,172.397,40.200,157.682
C08779=1046.428,311.352,-112.369,172.393,40.197,157.681
C08780=1046.420,311.105,-112.336,172.389,40.194,157.680
C08781=1046.413,310.857,-112.302,172.386,40.192,157.680
C08782=1046.406,310.609,-112.269,172.382,40.188,157.679
C08783=1046.399,310.361,-112.235,172.378,40.186,157.678
C08784=1046.392,310.114,-112.202,172.374,40.182,157.677
C08785=1046.386,309.866,-112.168,172.370,40.179,157.676
C08786=1046.379,309.619,-112.135,172.366,40.176,157.676
C08787=1046.372,309.371,-112.102,172.362,40.173,157.675
C08788=1046.365,309.123,-112.068,172.359,40.170,157.674
C08789=1046.358,308.876,-112.035,172.355,40.167,157.673
C08790=1046.351,308.628,-112.002,172.351,40.165,157.672
C08791=1046.343,308.381,-111.968,172.347,40.161,157.671
C08792=1046.337,308.133,-111.935,172.344,40.159,157.671
C08793=1046.330,307.885,-111.902,172.340,40.155,157.670
C08794=1046.324,307.638,-111.869,172.336,40.153,157.669
C08795=1046.316,307.390,-111.835,172.332,40.149,157.668
C08796=1046.310,307.142,-111.802,172.329,40.147,157.667
C08797=1046.303,306.895,-111.769,172.325,40.143,157.666
C08798=1046.297,306.647,-111.736,172.321,40.141,157.666
C08799=1046.289,306.400,-111.703,172.317,40.137,157.665
C08800=1046.282,306.152,-111.670,172.314,40.135,157.664
C08801=1046.276,305.904,-111.637,172.310,40.131,157.663
C08802=1046.269,305.657,-111.603,172.307,40.129,157.662
C08803=1046.260,305.347,-111.562,172.302,40.125,157.661
C08804=1046.252,305.036,-111.520,172.297,40.121,157.660
C08805=1046.244,304.727,-111.479,172.292,40.117,157.659
C08806=1046.235,304.416,-111.438,172.288,40.114,157.658
C08807=1046.228,304.168,-111.404,172.285,40.111,157.657
C08808=1046.222,303.921,-111.372,172.281,40.108,157.657
C08809=1046.215,303.673,-111.338,172.277,40.105,157.656
C08810=1046.207,303.426,-111.306,172.273,40.102,157.655
C08811=1046.201,303.178,-111.273,172.270,40.099,157.654
C08812=1046.194,302.930,-111.240,172.266,40.096,157.653
C08813=1046.188,302.682,-111.207,172.263,40.093,157.653
C08814=1046.181,302.434,-111.174,172.259,40.090,157.652
C08815=1046.175,302.187,-111.141,172.255,40.087,157.651
C08816=1046.167,301.940,-111.108,172.252,40.085,157.650
C08817=1046.160,301.692,-111.075,172.248,40.081,157.649
C08818=1046.154,301.444,-111.042,172.244,40.079,157.649
C08819=1046.148,301.196,-111.010,172.241,40.076,157.648
C08820=1046.141,300.948,-110.977,172.238,40.073,157.647
C08821=1046.134,300.701,-110.944,172.234,40.070,157.646
C08822=1046.128,300.453,-110.912,172.230,40.067,157.645
C08823=1046.121,300.205,-110.879,172.226,40.064,157.645
C08824=1046.114,299.957,-110.846,172.224,40.061,157.644
C08825=1046.108,299.710,-110.813,172.220,40.058,157.643
C08826=1046.102,299.462,-110.780,172.216,40.055,157.642
C08827=1046.094,299.214,-110.748,172.213,40.052,157.641
C08828=1046.088,298.967,-110.715,172.209,40.049,157.641
C08829=1046.082,298.719,-110.682,172.205,40.046,157.640
C08830=1046.075,298.471,-110.650,172.202,40.044,157.639
C08831=1046.068,298.223,-110.616,172.199,40.040,157.638
C08832=1046.061,297.976,-110.584,172.195,40.038,157.637
C08833=1046.055,297.728,-110.552,172.191,40.035,157.637
C08834=1046.049,297.481,-110.519,172.188,40.032,157.636
C08835=1046.042,297.232,-110.486,172.185,40.029,157.635
C08836=1046.035,296.985,-110.454,172.181,40.026,157.634
C08837=1046.029,296.738,-110.421,172.178,40.023,157.634
C08838=1046.023,296.489,-110.389,172.174,40.020,157.633
C08839=1046.016,296.242,-110.356,172.170,40.017,157.632
C08840=1046.010,295.994,-110.323,172.168,40.015,157.631
C08841=1046.002,295.746,-110.291,172.164,40.012,157.631
C08842=1045.996,295.498,-110.259,172.160,40.009,157.630
C08843=1045.989,295.251,-110.227,172.156,40.006,157.629
C08844=1045.983,295.003,-110.194,172.153,40.003,157.628
C08845=1045.976,294.754,-110.162,172.150,40.000,157.627
C08846=1045.969,294.507,-110.129,172.146,39.998,157.627
C08847=1045.962,294.260,-110.097,172.143,39.995,157.626
C08848=1045.956,294.012,-110.066,172.139,39.992,157.625
C08849=1045.949,293.764,-110.033,172.136,39.990,157.624
C08850=1045.943,293.516,-110.002,172.133,39.987,157.624
C08851=1045.936,293.268,-109.968,172.129,39.984,157.623
C08852=1045.929,293.021,-109.936,172.125,39.981,157.622
C08853=1045.922,292.773,-109.905,172.122,39.978,157.621
C08854=1045.916,292.525,-109.872,172.119,39.975,157.621
C08855=1045.909,292.277,-109.841,172.116,39.972,157.620
C08856=1045.902,292.029,-109.809,172.112,39.970,157.619
C08857=1045.895,291.781,-109.776,172.108,39.967,157.618
C08858=1045.889,291.533,-109.745,172.106,39.964,157.618
C08859=1045.881,291.240,-109.706,172.102,39.961,157.617
C08860=1045.873,290.946,-109.669,172.097,39.958,157.616
C08861=1045.865,290.652,-109.630,172.093,39.954,157.615
C08862=1045.857,290.358,-109.593,172.089,39.952,157.614
C08863=1045.850,290.110,-109.561,172.086,39.949,157.613
C08864=1045.844,289.862,-109.529,172.083,39.946,157.613
C08865=1045.837,289.615,-109.497,172.079,39.943,157.612
C08866=1045.831,289.367,-109.466,172.076,39.941,157.611
C08867=1045.824,289.119,-109.434,172.072,39.938,157.611
C08868=1045.818,288.871,-109.402,172.070,39.935,157.610
C08869=1045.811,288.623,-109.370,172.066,39.932,157.609
C08870=1045.804,288.375,-109.339,172.062,39.930,157.608
C08871=1045.797,288.128,-109.307,172.059,39.927,157.608
C08872=1045.791,287.880,-109.275,172.056,39.924,157.607
C08873=1045.784,287.632,-109.243,172.053,39.921,157.606
C08874=1045.778,287.384,-109.212,172.049,39.919,157.605
C08875=1045.771,287.136,-109.180,172.046,39.916,157.605
C08876=1045.764,286.889,-109.148,172.043,39.913,157.604
C08877=1045.757,286.641,-109.117,172.039,39.910,157.603
C08878=1045.750,286.393,-109.085,172.036,39.908,157.603
C08879=1045.744,286.145,-109.054,172.033,39.905,157.602
C08880=1045.737,285.897,-109.022,172.030,39.903,157.601
C08881=1045.730,285.649,-108.991,172.026,39.900,157.600
C08882=1045.724,285.401,-108.960,172.023,39.897,157.600
C08883=1045.718,285.153,-108.928,172.020,39.894,157.599
C08884=1045.711,284.905,-108.896,172.017,39.892,157.598
C08885=1045.704,284.657,-108.865,172.013,39.889,157.598
C08886=1045.697,284.410,-108.833,172.010,39.887,157.597
C08887=1045.691,284.162,-108.802,172.007,39.884,157.596
C08888=1045.684,283.914,-108.770,172.003,39.881,157.595
C08889=1045.677,283.666,-108.739,172.000,39.878,157.595
C08890=1045.671,283.418,-108.708,171.997,39.876,157.594
C08891=1045.664,283.170,-108.676,171.994,39.873,157.593
C08892=1045.657,282.922,-108.645,171.990,39.871,157.593
C08893=1045.651,282.674,-108.614,171.988,39.868,157.592
C08894=1045.644,282.426,-108.582,171.984,39.865,157.591
C08895=1045.637,282.178,-108.551,171.981,39.863,157.591
C08896=1045.630,281.930,-108.520,171.977,39.860,157.590
C08897=1045.624,281.682,-108.488,171.975,39.857,157.589
C08898=1045.618,281.435,-108.457,171.971,39.855,157.588
C08899=1045.611,281.186,-108.426,171.968,39.852,157.588
C08900=1045.605,280.938,-108.395,171.965,39.850,157.587
C08901=1045.598,280.690,-108.364,171.962,39.847,157.586
C08902=1045.591,280.443,-108.332,171.959,39.844,157.586
C08903=1045.585,280.194,-108.301,171.955,39.841,157.585
C08904=1045.579,279.947,-108.270,171.953,39.839,157.584
C08905=1045.572,279.699,-108.239,171.949,39.836,157.583
C08906=1045.565,279.451,-108.207,171.946,39.834,157.583
C08907=1045.559,279.203,-108.177,171.943,39.831,157.582
C08908=1045.552,278.955,-108.145,171.940,39.828,157.581
C08909=1045.545,278.707,-108.114,171.936,39.826,157.581
C08910=1045.539,278.459,-108.084,171.934,39.823,157.580
C08911=1045.532,278.211,-108.053,171.930,39.820,157.579
C08912=1045.525,277.963,-108.022,171.927,39.818,157.579
C08913=1045.519,277.715,-107.991,171.925,39.815,157.578
C08914=1045.512,277.467,-107.960,171.921,39.813,157.577
C08915=1045.504,277.185,-107.925,171.917,39.810,157.576
C08916=1045.497,276.903,-107.890,171.914,39.807,157.576
C08917=1045.490,276.621,-107.854,171.910,39.804,157.575
C08918=1045.482,276.338,-107.819,171.907,39.801,157.574
C08919=1045.475,276.091,-107.788,171.904,39.798,157.573
C08920=1045.469,275.842,-107.758,171.900,39.796,157.573
C08921=1045.462,275.594,-107.727,171.898,39.793,157.572
C08922=1045.455,275.346,-107.696,171.894,39.790,157.571
C08923=1045.449,275.098,-107.666,171.891,39.788,157.571
C08924=1045.443,274.851,-107.634,171.889,39.785,157.570
C08925=1045.435,274.602,-107.604,171.885,39.783,157.569
C08926=1045.429,274.354,-107.573,171.882,39.780,157.569
C08927=1045.423,274.107,-107.542,171.879,39.778,157.568
C08928=1045.416,273.858,-107.512,171.876,39.775,157.567
C08929=1045.409,273.610,-107.482,171.873,39.773,157.567
C08930=1045.403,273.362,-107.450,171.870,39.770,157.566
C08931=1045.396,273.114,-107.420,171.867,39.768,157.565
C08932=1045.390,272.866,-107.390,171.864,39.765,157.565
C08933=1045.383,272.618,-107.358,171.861,39.763,157.564
C08934=1045.376,272.371,-107.328,171.858,39.760,157.563
C08935=1045.370,272.122,-107.298,171.855,39.757,157.563
C08936=1045.363,271.873,-107.267,171.852,39.755,157.562
C08937=1045.357,271.627,-107.237,171.849,39.752,157.561
C08938=1045.350,271.378,-107.206,171.845,39.750,157.561
C08939=1045.343,271.130,-107.176,171.843,39.747,157.560
C08940=1045.337,270.882,-107.145,171.840,39.745,157.559
C08941=1045.330,270.634,-107.115,171.836,39.742,157.559
C08942=1045.324,270.385,-107.084,171.834,39.739,157.558
C08943=1045.317,270.138,-107.054,171.831,39.737,157.557
C08944=1045.310,269.890,-107.023,171.827,39.734,157.557
C08945=1045.303,269.642,-106.993,171.825,39.732,157.556
C08946=1045.297,269.394,-106.963,171.822,39.729,157.555
C08947=1045.290,269.146,-106.933,171.818,39.727,157.555
C08948=1045.284,268.897,-106.902,171.816,39.724,157.554
C08949=1045.277,268.650,-106.872,171.813,39.722,157.553
C08950=1045.271,268.401,-106.842,171.809,39.719,157.553
C08951=1045.264,268.154,-106.812,171.807,39.717,157.552
C08952=1045.258,267.905,-106.781,171.804,39.714,157.551
C08953=1045.251,267.657,-106.751,171.801,39.712,157.551
C08954=1045.245,267.409,-106.721,171.798,39.709,157.550
C08955=1045.238,267.161,-106.690,171.795,39.707,157.550
C08956=1045.231,266.913,-106.661,171.792,39.704,157.549
C08957=1045.225,266.665,-106.630,171.789,39.702,157.548
C08958=1045.218,266.417,-106.600,171.786,39.699,157.548
C08959=1045.211,266.169,-106.570,171.784,39.697,157.547
C08960=1045.205,265.920,-106.540,171.780,39.694,157.546
C08961=1045.198,265.672,-106.510,171.777,39.692,157.546
C08962=1045.191,265.424,-106.480,171.775,39.689,157.545
C08963=1045.185,265.176,-106.450,171.772,39.687,157.544
C08964=1045.178,264.928,-106.420,171.768,39.684,157.544
C08965=1045.172,264.681,-106.390,171.766,39.682,157.543
C08966=1045.166,264.431,-106.360,171.763,39.679,157.542
C08967=1045.158,264.183,-106.330,171.760,39.677,157.542
C08968=1045.152,263.936,-106.300,171.757,39.674,157.541
C08969=1045.145,263.687,-106.269,171.754,39.672,157.540
C08970=1045.139,263.439,-106.240,171.751,39.669,157.540
C08971=1045.132,263.162,-106.207,171.748,39.667,157.539
C08972=1045.124,262.884,-106.173,171.745,39.664,157.538
C08973=1045.117,262.606,-106.140,171.741,39.661,157.538
C08974=1045.110,262.328,-106.106,171.739,39.658,157.537
C08975=1045.103,262.080,-106.076,171.736,39.655,157.536
C08976=1045.097,261.832,-106.047,171.732,39.653,157.536
C08977=1045.090,261.584,-106.017,171.730,39.651,157.535
C08978=1045.083,261.335,-105.988,171.727,39.649,157.535
C08979=1045.076,261.088,-105.958,171.724,39.646,157.534
C08980=1045.069,260.839,-105.928,171.721,39.644,157.533
C08981=1045.063,260.591,-105.899,171.718,39.641,157.533
C08982=1045.056,260.343,-105.869,171.716,39.639,157.532
C08983=1045.049,260.095,-105.839,171.713,39.636,157.531
C08984=1045.042,259.847,-105.809,171.709,39.634,157.531
C08985=1045.036,259.599,-105.780,171.707,39.631,157.530
C08986=1045.028,259.351,-105.751,171.704,39.629,157.529
C08987=1045.022,259.103,-105.722,171.702,39.627,157.529
C08988=1045.016,258.854,-105.693,171.699,39.625,157.528
C08989=1045.008,258.606,-105.663,171.695,39.622,157.528
C08990=1045.002,258.358,-105.634,171.693,39.620,157.527
C08991=1044.995,258.110,-105.603,171.690,39.617,157.526
C08992=1044.989,257.862,-105.574,171.688,39.614,157.526
C08993=1044.982,257.613,-105.545,171.685,39.612,157.525
C08994=1044.975,257.365,-105.515,171.681,39.610,157.525
C08995=1044.969,257.117,-105.486,171.679,39.607,157.524
C08996=1044.962,256.868,-105.457,171.676,39.605,157.523
C08997=1044.956,256.621,-105.427,171.674,39.603,157.523
C08998=1044.949,256.372,-105.398,171.671,39.600,157.522
C08999=1044.943,256.124,-105.369,171.667,39.598,157.521
C09000=1044.935,255.876,-105.338,171.665,39.595,157.521
C09001=1044.929,255.628,-105.309,171.662,39.593,157.520
C09002=1044.922,255.380,-105.281,171.659,39.590,157.520
C09003=1044.915,255.132,-105.251,171.657,39.588,157.519
C09004=1044.909,254.883,-105.222,171.654,39.586,157.518
C09005=1044.903,254.635,-105.193,171.652,39.583,157.518
C09006=1044.896,254.386,-105.163,171.648,39.581,157.517
C09007=1044.889,254.139,-105.134,171.645,39.578,157.517
C09008=1044.883,253.891,-105.105,171.643,39.576,157.516
C09009=1044.876,253.642,-105.075,171.640,39.573,157.515
C09010=1044.870,253.394,-105.046,171.638,39.571,157.515
C09011=1044.864,253.146,-105.017,171.635,39.568,157.514
C09012=1044.857,252.897,-104.988,171.632,39.566,157.513
C09013=1044.850,252.649,-104.958,171.630,39.564,157.513
C09014=1044.843,252.402,-104.929,171.626,39.561,157.512
C09015=1044.837,252.153,-104.900,171.624,39.559,157.512
C09016=1044.830,251.905,-104.871,171.621,39.556,157.511
C09017=1044.824,251.656,-104.842,171.618,39.554,157.510
C09018=1044.818,251.408,-104.813,171.616,39.551,157.510
C09019=1044.811,251.159,-104.784,171.613,39.549,157.509
C09020=1044.805,250.911,-104.754,171.610,39.546,157.508
C09021=1044.798,250.663,-104.725,171.608,39.544,157.508
C09022=1044.792,250.415,-104.696,171.605,39.542,157.507
C09023=1044.785,250.167,-104.668,171.603,39.539,157.507
C09024=1044.778,249.918,-104.639,171.600,39.537,157.506
C09025=1044.772,249.671,-104.609,171.597,39.534,157.505
C09026=1044.765,249.423,-104.580,171.594,39.531,157.505
C09027=1044.758,249.143,-104.548,171.591,39.529,157.504
C09028=1044.752,248.864,-104.515,171.589,39.526,157.503
C09029=1044.744,248.585,-104.482,171.586,39.523,157.503
C09030=1044.737,248.306,-104.450,171.582,39.521,157.502
C09031=1044.730,248.058,-104.420,171.580,39.518,157.501
C09032=1044.724,247.809,-104.391,171.577,39.516,157.501
C09033=1044.717,247.561,-104.362,171.574,39.513,157.500
C09034=1044.710,247.313,-104.334,171.572,39.511,157.500
C09035=1044.704,247.065,-104.305,171.569,39.508,157.499
C09036=1044.698,246.816,-104.276,171.567,39.506,157.498
C09037=1044.692,246.568,-104.247,171.564,39.503,157.498
